DECL E6POS XP287={X 5671.46198,Y -717.1018,Z 4003.704,A -116.65787,B -23.21109,C 16.21129,S 2,T 35,E1 -3867.99764,E2 0,E3 0,E4 0,E5 0,E6 0}
; DECL LDAT LCPDATP147={VEL 1,ACC 100,APO_DIST 100,APO_FAC 50.0,ORI_TYP #VAR,CIRC_TYP #BASE,JERK_FAC 50.0}
DECL FDAT FP288={TOOL_NO 0,BASE_NO 0,IPO_FRAME #BASE,POINT2[] " ",TQ_STATE FALSE}
DECL E6POS XP288={X 12666.37592,Y -538.48386,Z 3708.53974,A -127.07895,B -20.60151,C -3.44033,S 2,T 35,E1 -10812.08896,E2 0,E3 0,E4 0,E5 0,E6 0}
; DECL LDAT LCPDATP113={VEL 1,ACC 100,APO_DIST 100,APO_FAC 50.0,ORI_TYP #VAR,CIRC_TYP #BASE,JERK_FAC 50.0}
DECL FDAT FP289={TOOL_NO 0,BASE_NO 0,IPO_FRAME #BASE,POINT2[] " ",TQ_STATE FALSE}
DECL E6POS XP289={X 6379.94734,Y -681.40788,Z 3158.20554,A -102.40256,B 11.37187,C 4.81103,S 2,T 35,E1 -4209.91162,E2 0,E3 0,E4 0,E5 0,E6 0}
; DECL LDAT LCPDATP114={VEL 1,ACC 100,APO_DIST 100,APO_FAC 50.0,ORI_TYP #VAR,CIRC_TYP #BASE,JERK_FAC 50.0}
DECL FDAT FP290={TOOL_NO 0,BASE_NO 0,IPO_FRAME #BASE,POINT2[] " ",TQ_STATE FALSE}
DECL E6POS XP290={X 6328.481,Y -681.40737,Z 3158.20597,A -102.7078,B 7.77597,C 4.76025,S 2,T 35,E1 -4158.44503,E2 0,E3 0,E4 0,E5 0,E6 0}
; DECL LDAT LCPDATP115={VEL 1,ACC 100,APO_DIST 100,APO_FAC 50.0,ORI_TYP #VAR,CIRC_TYP #BASE,JERK_FAC 50.0}
DECL FDAT FP291={TOOL_NO 0,BASE_NO 0,IPO_FRAME #BASE,POINT2[] " ",TQ_STATE FALSE}
DECL E6POS XP291={X 12929.38089,Y -681.40737,Z 3158.20639,A -83.4604,B -12.81532,C -0.94267,S 2,T 35,E1 -10812.08896,E2 0,E3 0,E4 0,E5 0,E6 0}
; DECL LDAT LCPDATP116={VEL 1,ACC 100,APO_DIST 100,APO_FAC 50.0,ORI_TYP #VAR,CIRC_TYP #BASE,JERK_FAC 50.0}
DECL FDAT FP292={TOOL_NO 0,BASE_NO 0,IPO_FRAME #BASE,POINT2[] " ",TQ_STATE FALSE}
DECL E6POS XP292={X 12886.08572,Y -646.4113,Z 3336.02814,A -83.4604,B -12.81532,C -0.94267,S 2,T 35,E1 -10812.08896,E2 0,E3 0,E4 0,E5 0,E6 0}
; DECL LDAT LCPDATP117={VEL 1,ACC 100,APO_DIST 100,APO_FAC 50.0,ORI_TYP #VAR,CIRC_TYP #BASE,JERK_FAC 50.0}
DECL FDAT FP293={TOOL_NO 0,BASE_NO 0,IPO_FRAME #BASE,POINT2[] " ",TQ_STATE FALSE}
DECL E6POS XP293={X 6226.20694,Y -691.76303,Z 3410.82553,A -102.7078,B 7.77597,C 4.76022,S 2,T 35,E1 -4167.06683,E2 0,E3 0,E4 0,E5 0,E6 0}
; DECL LDAT LCPDATP118={VEL 1,ACC 100,APO_DIST 100,APO_FAC 50.0,ORI_TYP #VAR,CIRC_TYP #BASE,JERK_FAC 50.0}
DECL FDAT FP294={TOOL_NO 0,BASE_NO 0,IPO_FRAME #BASE,POINT2[] " ",TQ_STATE FALSE}
DECL E6POS XP294={X 6109.20944,Y -705.3695,Z 3654.40552,A -102.70779,B 7.77597,C 4.76025,S 2,T 35,E1 -4140.9372,E2 0,E3 0,E4 0,E5 0,E6 0}
; DECL LDAT LCPDATP121={VEL 1,ACC 100,APO_DIST 100,APO_FAC 50.0,ORI_TYP #VAR,CIRC_TYP #BASE,JERK_FAC 50.0}
DECL FDAT FP295={TOOL_NO 0,BASE_NO 0,IPO_FRAME #BASE,POINT2[] " ",TQ_STATE FALSE}
DECL E6POS XP295={X 12777.06723,Y -602.17839,Z 3573.69413,A -83.4604,B -12.81532,C -0.94267,S 2,T 35,E1 -10812.08896,E2 0,E3 0,E4 0,E5 0,E6 0}
; DECL LDAT LCPDATP122={VEL 1,ACC 100,APO_DIST 100,APO_FAC 50.0,ORI_TYP #VAR,CIRC_TYP #BASE,JERK_FAC 50.0}
DECL FDAT FP296={TOOL_NO 0,BASE_NO 0,IPO_FRAME #BASE,POINT2[] " ",TQ_STATE FALSE}
DECL E6POS XP296={X 12675.92788,Y -569.18264,Z 3775.2407,A -83.4604,B -12.81532,C -0.94267,S 2,T 35,E1 -10812.08896,E2 0,E3 0,E4 0,E5 0,E6 0}
; DECL LDAT LCPDATP119={VEL 1,ACC 100,APO_DIST 100,APO_FAC 50.0,ORI_TYP #VAR,CIRC_TYP #BASE,JERK_FAC 50.0}
DECL FDAT FP297={TOOL_NO 0,BASE_NO 0,IPO_FRAME #BASE,POINT2[] " ",TQ_STATE FALSE}
DECL E6POS XP297={X 6034.81499,Y -708.12179,Z 3847.76366,A -102.7078,B 7.77596,C 4.76026,S 2,T 35,E1 -4174.36752,E2 0,E3 0,E4 0,E5 0,E6 0}
; DECL LDAT LCPDATP120={VEL 1,ACC 100,APO_DIST 100,APO_FAC 50.0,ORI_TYP #VAR,CIRC_TYP #BASE,JERK_FAC 50.0}
DECL FDAT FP298={TOOL_NO 0,BASE_NO 0,IPO_FRAME #BASE,POINT2[] " ",TQ_STATE FALSE}
DECL E6POS XP298={X 5808.56571,Y -717.10091,Z 4003.7046,A -102.70779,B 7.77596,C 4.76025,S 2,T 35,E1 -4005.10214,E2 0,E3 0,E4 0,E5 0,E6 0}
; DECL LDAT LCPDATP123={VEL 1,ACC 100,APO_DIST 100,APO_FAC 50.0,ORI_TYP #VAR,CIRC_TYP #BASE,JERK_FAC 50.0}
DECL FDAT FP299={TOOL_NO 0,BASE_NO 0,IPO_FRAME #BASE,POINT2[] " ",TQ_STATE FALSE}
DECL E6POS XP299={X 12607.03936,Y -538.48386,Z 3940.5062,A -83.4604,B -12.81532,C -0.94267,S 2,T 35,E1 -10812.08896,E2 0,E3 0,E4 0,E5 0,E6 0}
; DECL LDAT LCPDATP124={VEL 1,ACC 100,APO_DIST 100,APO_FAC 50.0,ORI_TYP #VAR,CIRC_TYP #BASE,JERK_FAC 50.0}
DECL FDAT FP300={TOOL_NO 0,BASE_NO 0,IPO_FRAME #BASE,POINT2[] " ",TQ_STATE FALSE}
DECL E6POS XP300={X 12329.73693,Y -538.48386,Z 3940.5062,A -83.38777,B -15.32829,C -1.2413,S 2,T 35,E1 -10812.08896,E2 0,E3 0,E4 0,E5 0,E6 0}
; DECL LDAT LCPDATP130={VEL 1,ACC 100,APO_DIST 100,APO_FAC 50.0,ORI_TYP #VAR,CIRC_TYP #BASE,JERK_FAC 50.0}
DECL FDAT FP301={TOOL_NO 0,BASE_NO 0,IPO_FRAME #BASE,POINT2[] " ",TQ_STATE FALSE}
DECL E6POS XP301={X 6035.27715,Y -717.10158,Z 4003.70466,A -106.51042,B 6.34838,C 5.00917,S 2,T 35,E1 -4231.81368,E2 0,E3 0,E4 0,E5 0,E6 0}
; DECL LDAT LCPDATP131={VEL 1,ACC 100,APO_DIST 100,APO_FAC 50.0,ORI_TYP #VAR,CIRC_TYP #BASE,JERK_FAC 50.0}
DECL FDAT FP302={TOOL_NO 0,BASE_NO 0,IPO_FRAME #BASE,POINT2[] " ",TQ_STATE FALSE}
DECL E6POS XP302={X 6001.84737,Y -717.10113,Z 4003.70421,A -106.4599,B 4.5615,C 5.54032,S 2,T 35,E1 -4198.38336,E2 0,E3 0,E4 0,E5 0,E6 0}
; DECL LDAT LCPDATP125={VEL 1,ACC 100,APO_DIST 100,APO_FAC 50.0,ORI_TYP #VAR,CIRC_TYP #BASE,JERK_FAC 50.0}
DECL FDAT FP303={TOOL_NO 0,BASE_NO 0,IPO_FRAME #BASE,POINT2[] " ",TQ_STATE FALSE}
DECL E6POS XP303={X 12327.62864,Y -538.48366,Z 3940.50597,A -87.76623,B -17.49847,C -1.50503,S 2,T 35,E1 -10473.34117,E2 0,E3 0,E4 0,E5 0,E6 0}
; DECL LDAT LCPDATP126={VEL 1,ACC 100,APO_DIST 100,APO_FAC 50.0,ORI_TYP #VAR,CIRC_TYP #BASE,JERK_FAC 50.0}
DECL FDAT FP304={TOOL_NO 0,BASE_NO 0,IPO_FRAME #BASE,POINT2[] " ",TQ_STATE FALSE}
DECL E6POS XP304={X 12344.44126,Y -538.48354,Z 3940.50612,A -92.12133,B -19.55447,C -1.59012,S 2,T 35,E1 -10490.15446,E2 0,E3 0,E4 0,E5 0,E6 0}
; DECL LDAT LCPDATP132={VEL 1,ACC 100,APO_DIST 100,APO_FAC 50.0,ORI_TYP #VAR,CIRC_TYP #BASE,JERK_FAC 50.0}
DECL FDAT FP305={TOOL_NO 0,BASE_NO 0,IPO_FRAME #BASE,POINT2[] " ",TQ_STATE FALSE}
DECL E6POS XP305={X 5984.60315,Y -717.10142,Z 4003.7045,A -107.27293,B 2.66443,C 6.10126,S 2,T 35,E1 -4181.13976,E2 0,E3 0,E4 0,E5 0,E6 0}
; DECL LDAT LCPDATP133={VEL 1,ACC 100,APO_DIST 100,APO_FAC 50.0,ORI_TYP #VAR,CIRC_TYP #BASE,JERK_FAC 50.0}
DECL FDAT FP306={TOOL_NO 0,BASE_NO 0,IPO_FRAME #BASE,POINT2[] " ",TQ_STATE FALSE}
DECL E6POS XP306={X 5959.53065,Y -717.10165,Z 4003.70439,A -107.25516,B 0.74219,C 6.69889,S 2,T 35,E1 -4156.06702,E2 0,E3 0,E4 0,E5 0,E6 0}
; DECL LDAT LCPDATP127={VEL 1,ACC 100,APO_DIST 100,APO_FAC 50.0,ORI_TYP #VAR,CIRC_TYP #BASE,JERK_FAC 50.0}
DECL FDAT FP307={TOOL_NO 0,BASE_NO 0,IPO_FRAME #BASE,POINT2[] " ",TQ_STATE FALSE}
DECL E6POS XP307={X 12327.65948,Y -538.48376,Z 3940.50627,A -96.02004,B -21.56802,C -1.50992,S 2,T 35,E1 -10473.37259,E2 0,E3 0,E4 0,E5 0,E6 0}
; DECL LDAT LCPDATP128={VEL 1,ACC 100,APO_DIST 100,APO_FAC 50.0,ORI_TYP #VAR,CIRC_TYP #BASE,JERK_FAC 50.0}
DECL FDAT FP308={TOOL_NO 0,BASE_NO 0,IPO_FRAME #BASE,POINT2[] " ",TQ_STATE FALSE}
DECL E6POS XP308={X 12434.40962,Y -538.48361,Z 3791.38491,A -100.48203,B -23.59142,C -1.27711,S 2,T 35,E1 -10580.12251,E2 0,E3 0,E4 0,E5 0,E6 0}
; DECL LDAT LCPDATP134={VEL 1,ACC 100,APO_DIST 100,APO_FAC 50.0,ORI_TYP #VAR,CIRC_TYP #BASE,JERK_FAC 50.0}
DECL FDAT FP309={TOOL_NO 0,BASE_NO 0,IPO_FRAME #BASE,POINT2[] " ",TQ_STATE FALSE}
DECL E6POS XP309={X 6027.18413,Y -717.10157,Z 4003.70451,A -108.83879,B -1.2655,C 7.3225,S 2,T 35,E1 -4223.72032,E2 0,E3 0,E4 0,E5 0,E6 0}
; DECL LDAT LCPDATP135={VEL 1,ACC 100,APO_DIST 100,APO_FAC 50.0,ORI_TYP #VAR,CIRC_TYP #BASE,JERK_FAC 50.0}
DECL FDAT FP310={TOOL_NO 0,BASE_NO 0,IPO_FRAME #BASE,POINT2[] " ",TQ_STATE FALSE}
DECL E6POS XP310={X 5994.01853,Y -717.10159,Z 4003.70409,A -109.42003,B -3.44272,C 8.06654,S 2,T 35,E1 -4190.55423,E2 0,E3 0,E4 0,E5 0,E6 0}
; DECL LDAT LCPDATP129={VEL 1,ACC 100,APO_DIST 100,APO_FAC 50.0,ORI_TYP #VAR,CIRC_TYP #BASE,JERK_FAC 50.0}
DECL FDAT FP311={TOOL_NO 0,BASE_NO 0,IPO_FRAME #BASE,POINT2[] " ",TQ_STATE FALSE}
DECL E6POS XP311={X 12525.53957,Y -538.48385,Z 3733.39322,A -103.74147,B -24.12805,C -1.24549,S 2,T 35,E1 -10671.25219,E2 0,E3 0,E4 0,E5 0,E6 0}
; DECL LDAT LCPDATP138={VEL 1,ACC 100,APO_DIST 100,APO_FAC 50.0,ORI_TYP #VAR,CIRC_TYP #BASE,JERK_FAC 50.0}
DECL FDAT FP312={TOOL_NO 0,BASE_NO 0,IPO_FRAME #BASE,POINT2[] " ",TQ_STATE FALSE}
DECL E6POS XP312={X 12409.55634,Y -538.48385,Z 3733.39322,A -103.74147,B -24.12805,C -1.24549,S 2,T 35,E1 -10555.26896,E2 0,E3 0,E4 0,E5 0,E6 0}
; DECL LDAT LCPDATP136={VEL 1,ACC 100,APO_DIST 100,APO_FAC 50.0,ORI_TYP #VAR,CIRC_TYP #BASE,JERK_FAC 50.0}
DECL FDAT FP313={TOOL_NO 0,BASE_NO 0,IPO_FRAME #BASE,POINT2[] " ",TQ_STATE FALSE}
DECL E6POS XP313={X 5960.30101,Y -717.10136,Z 4003.70387,A -109.95564,B -5.51238,C 8.79955,S 2,T 35,E1 -4156.83652,E2 0,E3 0,E4 0,E5 0,E6 0}
; DECL LDAT LCPDATP137={VEL 1,ACC 100,APO_DIST 100,APO_FAC 50.0,ORI_TYP #VAR,CIRC_TYP #BASE,JERK_FAC 50.0}
DECL FDAT FP314={TOOL_NO 0,BASE_NO 0,IPO_FRAME #BASE,POINT2[] " ",TQ_STATE FALSE}
DECL E6POS XP314={X 5959.29294,Y -717.10098,Z 4003.70454,A -110.58224,B -7.77816,C 9.62993,S 2,T 35,E1 -4155.82897,E2 0,E3 0,E4 0,E5 0,E6 0}
; DECL LDAT LCPDATP139={VEL 1,ACC 100,APO_DIST 100,APO_FAC 50.0,ORI_TYP #VAR,CIRC_TYP #BASE,JERK_FAC 50.0}
DECL FDAT FP315={TOOL_NO 0,BASE_NO 0,IPO_FRAME #BASE,POINT2[] " ",TQ_STATE FALSE}
DECL E6POS XP315={X 12666.37592,Y -538.48386,Z 3733.39329,A -110.95703,B -23.34196,C -1.63568,S 2,T 35,E1 -10812.08896,E2 0,E3 0,E4 0,E5 0,E6 0}
; DECL LDAT LCPDATP140={VEL 1,ACC 100,APO_DIST 100,APO_FAC 50.0,ORI_TYP #VAR,CIRC_TYP #BASE,JERK_FAC 50.0}
DECL FDAT FP316={TOOL_NO 0,BASE_NO 0,IPO_FRAME #BASE,POINT2[] " ",TQ_STATE FALSE}
DECL E6POS XP316={X 12666.37592,Y -538.48386,Z 3700.25522,A -113.36831,B -23.34196,C -1.63568,S 2,T 35,E1 -10812.08896,E2 0,E3 0,E4 0,E5 0,E6 0}
; DECL LDAT LCPDATP149={VEL 1,ACC 100,APO_DIST 100,APO_FAC 50.0,ORI_TYP #VAR,CIRC_TYP #BASE,JERK_FAC 50.0}
DECL FDAT FP317={TOOL_NO 0,BASE_NO 0,IPO_FRAME #BASE,POINT2[] " ",TQ_STATE FALSE}
DECL E6POS XP317={X 5916.8006,Y -717.10155,Z 4003.70412,A -110.72224,B -10.13455,C 10.52896,S 2,T 35,E1 -4113.33656,E2 0,E3 0,E4 0,E5 0,E6 0}
; DECL LDAT LCPDATP150={VEL 1,ACC 100,APO_DIST 100,APO_FAC 50.0,ORI_TYP #VAR,CIRC_TYP #BASE,JERK_FAC 50.0}
DECL FDAT FP318={TOOL_NO 0,BASE_NO 0,IPO_FRAME #BASE,POINT2[] " ",TQ_STATE FALSE}
DECL E6POS XP318={X 5875.31565,Y -717.1012,Z 4003.70448,A -110.8879,B -12.32973,C 11.37928,S 2,T 35,E1 -4071.85169,E2 0,E3 0,E4 0,E5 0,E6 0}
; DECL LDAT LCPDATP141={VEL 1,ACC 100,APO_DIST 100,APO_FAC 50.0,ORI_TYP #VAR,CIRC_TYP #BASE,JERK_FAC 50.0}
DECL FDAT FP319={TOOL_NO 0,BASE_NO 0,IPO_FRAME #BASE,POINT2[] " ",TQ_STATE FALSE}
DECL E6POS XP319={X 12666.37592,Y -538.48386,Z 3675.40167,A -115.34787,B -23.34196,C -1.63568,S 2,T 35,E1 -10812.08896,E2 0,E3 0,E4 0,E5 0,E6 0}
; DECL LDAT LCPDATP142={VEL 1,ACC 100,APO_DIST 100,APO_FAC 50.0,ORI_TYP #VAR,CIRC_TYP #BASE,JERK_FAC 50.0}
DECL FDAT FP320={TOOL_NO 0,BASE_NO 0,IPO_FRAME #BASE,POINT2[] " ",TQ_STATE FALSE}
DECL E6POS XP320={X 12666.37592,Y -538.48386,Z 3725.10877,A -117.62399,B -22.31862,C -2.21953,S 2,T 35,E1 -10812.08896,E2 0,E3 0,E4 0,E5 0,E6 0}
; DECL LDAT LCPDATP151={VEL 1,ACC 100,APO_DIST 100,APO_FAC 50.0,ORI_TYP #VAR,CIRC_TYP #BASE,JERK_FAC 50.0}
DECL FDAT FP321={TOOL_NO 0,BASE_NO 0,IPO_FRAME #BASE,POINT2[] " ",TQ_STATE FALSE}
DECL E6POS XP321={X 5898.57722,Y -717.10122,Z 4003.70435,A -112.09203,B -14.38754,C 12.19033,S 2,T 35,E1 -4095.11298,E2 0,E3 0,E4 0,E5 0,E6 0}
; DECL LDAT LCPDATP152={VEL 1,ACC 100,APO_DIST 100,APO_FAC 50.0,ORI_TYP #VAR,CIRC_TYP #BASE,JERK_FAC 50.0}
DECL FDAT FP322={TOOL_NO 0,BASE_NO 0,IPO_FRAME #BASE,POINT2[] " ",TQ_STATE FALSE}
DECL E6POS XP322={X 5854.40488,Y -717.10171,Z 4003.70448,A -112.35649,B -16.71303,C 13.17652,S 2,T 35,E1 -4050.94133,E2 0,E3 0,E4 0,E5 0,E6 0}
; DECL LDAT LCPDATP143={VEL 1,ACC 100,APO_DIST 100,APO_FAC 50.0,ORI_TYP #VAR,CIRC_TYP #BASE,JERK_FAC 50.0}
DECL FDAT FP323={TOOL_NO 0,BASE_NO 0,IPO_FRAME #BASE,POINT2[] " ",TQ_STATE FALSE}
DECL E6POS XP323={X 12666.37592,Y -538.48386,Z 3708.53974,A -119.39266,B -22.0406,C -2.38888,S 2,T 35,E1 -10812.08896,E2 0,E3 0,E4 0,E5 0,E6 0}
; DECL LDAT LCPDATP144={VEL 1,ACC 100,APO_DIST 100,APO_FAC 50.0,ORI_TYP #VAR,CIRC_TYP #BASE,JERK_FAC 50.0}
DECL FDAT FP324={TOOL_NO 0,BASE_NO 0,IPO_FRAME #BASE,POINT2[] " ",TQ_STATE FALSE}
DECL E6POS XP324={X 12666.37592,Y -538.48386,Z 3716.82426,A -121.52366,B -21.70131,C -2.61349,S 2,T 35,E1 -10812.08896,E2 0,E3 0,E4 0,E5 0,E6 0}
; DECL LDAT LCPDATP153={VEL 1,ACC 100,APO_DIST 100,APO_FAC 50.0,ORI_TYP #VAR,CIRC_TYP #BASE,JERK_FAC 50.0}
DECL FDAT FP325={TOOL_NO 0,BASE_NO 0,IPO_FRAME #BASE,POINT2[] " ",TQ_STATE FALSE}
DECL E6POS XP325={X 5865.70091,Y -717.10124,Z 4003.70383,A -113.62634,B -18.80667,C 14.08679,S 2,T 35,E1 -4062.23613,E2 0,E3 0,E4 0,E5 0,E6 0}
; DECL LDAT LCPDATP154={VEL 1,ACC 100,APO_DIST 100,APO_FAC 50.0,ORI_TYP #VAR,CIRC_TYP #BASE,JERK_FAC 50.0}
DECL FDAT FP326={TOOL_NO 0,BASE_NO 0,IPO_FRAME #BASE,POINT2[] " ",TQ_STATE FALSE}
DECL E6POS XP326={X 5786.97193,Y -717.10138,Z 4003.70442,A -113.90846,B -20.59534,C 14.92344,S 2,T 35,E1 -3983.50839,E2 0,E3 0,E4 0,E5 0,E6 0}
; DECL LDAT LCPDATP145={VEL 1,ACC 100,APO_DIST 100,APO_FAC 50.0,ORI_TYP #VAR,CIRC_TYP #BASE,JERK_FAC 50.0}
DECL FDAT FP327={TOOL_NO 0,BASE_NO 0,IPO_FRAME #BASE,POINT2[] " ",TQ_STATE FALSE}
DECL E6POS XP327={X 12666.37592,Y -538.48386,Z 3691.97071,A -122.58569,B -21.70131,C -2.61349,S 2,T 35,E1 -10812.08896,E2 0,E3 0,E4 0,E5 0,E6 0}
; DECL LDAT LCPDATP146={VEL 1,ACC 100,APO_DIST 100,APO_FAC 50.0,ORI_TYP #VAR,CIRC_TYP #BASE,JERK_FAC 50.0}
DECL FDAT FP328={TOOL_NO 0,BASE_NO 0,IPO_FRAME #BASE,POINT2[] " ",TQ_STATE FALSE}
DECL E6POS XP328={X 12666.37592,Y -538.48386,Z 3741.67781,A -124.88801,B -20.60151,C -3.44033,S 2,T 35,E1 -10812.08896,E2 0,E3 0,E4 0,E5 0,E6 0}
; DECL LDAT LCPDATP155={VEL 1,ACC 100,APO_DIST 100,APO_FAC 50.0,ORI_TYP #VAR,CIRC_TYP #BASE,JERK_FAC 50.0}
DECL FDAT FP329={TOOL_NO 0,BASE_NO 0,IPO_FRAME #BASE,POINT2[] " ",TQ_STATE FALSE}
DECL E6POS XP329={X 5766.06143,Y -717.10078,Z 4003.7047,A -114.88478,B -21.82725,C 15.51221,S 2,T 35,E1 -3962.59803,E2 0,E3 0,E4 0,E5 0,E6 0}
; DECL LDAT LCPDATP156={VEL 1,ACC 100,APO_DIST 100,APO_FAC 50.0,ORI_TYP #VAR,CIRC_TYP #BASE,JERK_FAC 50.0}
DECL FDAT FP330={TOOL_NO 0,BASE_NO 0,IPO_FRAME #BASE,POINT2[] " ",TQ_STATE FALSE}
DECL E6POS XP330={X 5671.46198,Y -717.1018,Z 4003.704,A -116.65787,B -23.21109,C 16.21129,S 2,T 35,E1 -3867.99764,E2 0,E3 0,E4 0,E5 0,E6 0}
; DECL LDAT LCPDATP147={VEL 1,ACC 100,APO_DIST 100,APO_FAC 50.0,ORI_TYP #VAR,CIRC_TYP #BASE,JERK_FAC 50.0}
DECL FDAT FP331={TOOL_NO 0,BASE_NO 0,IPO_FRAME #BASE,POINT2[] " ",TQ_STATE FALSE}
DECL E6POS XP331={X 12666.37592,Y -538.48386,Z 3708.53974,A -127.07895,B -20.60151,C -3.44033,S 2,T 35,E1 -10812.08896,E2 0,E3 0,E4 0,E5 0,E6 0}
; DECL LDAT LCPDATP113={VEL 1,ACC 100,APO_DIST 100,APO_FAC 50.0,ORI_TYP #VAR,CIRC_TYP #BASE,JERK_FAC 50.0}
DECL FDAT FP332={TOOL_NO 0,BASE_NO 0,IPO_FRAME #BASE,POINT2[] " ",TQ_STATE FALSE}
DECL E6POS XP332={X 6379.94734,Y -681.40788,Z 3158.20554,A -102.40256,B 11.37187,C 4.81103,S 2,T 35,E1 -4209.91162,E2 0,E3 0,E4 0,E5 0,E6 0}
; DECL LDAT LCPDATP114={VEL 1,ACC 100,APO_DIST 100,APO_FAC 50.0,ORI_TYP #VAR,CIRC_TYP #BASE,JERK_FAC 50.0}
DECL FDAT FP333={TOOL_NO 0,BASE_NO 0,IPO_FRAME #BASE,POINT2[] " ",TQ_STATE FALSE}
DECL E6POS XP333={X 6328.481,Y -681.40737,Z 3158.20597,A -102.7078,B 7.77597,C 4.76025,S 2,T 35,E1 -4158.44503,E2 0,E3 0,E4 0,E5 0,E6 0}
; DECL LDAT LCPDATP115={VEL 1,ACC 100,APO_DIST 100,APO_FAC 50.0,ORI_TYP #VAR,CIRC_TYP #BASE,JERK_FAC 50.0}
DECL FDAT FP334={TOOL_NO 0,BASE_NO 0,IPO_FRAME #BASE,POINT2[] " ",TQ_STATE FALSE}
DECL E6POS XP334={X 12929.38089,Y -681.40737,Z 3158.20639,A -83.4604,B -12.81532,C -0.94267,S 2,T 35,E1 -10812.08896,E2 0,E3 0,E4 0,E5 0,E6 0}
; DECL LDAT LCPDATP116={VEL 1,ACC 100,APO_DIST 100,APO_FAC 50.0,ORI_TYP #VAR,CIRC_TYP #BASE,JERK_FAC 50.0}
DECL FDAT FP335={TOOL_NO 0,BASE_NO 0,IPO_FRAME #BASE,POINT2[] " ",TQ_STATE FALSE}
DECL E6POS XP335={X 12886.08572,Y -646.4113,Z 3336.02814,A -83.4604,B -12.81532,C -0.94267,S 2,T 35,E1 -10812.08896,E2 0,E3 0,E4 0,E5 0,E6 0}
; DECL LDAT LCPDATP117={VEL 1,ACC 100,APO_DIST 100,APO_FAC 50.0,ORI_TYP #VAR,CIRC_TYP #BASE,JERK_FAC 50.0}
DECL FDAT FP336={TOOL_NO 0,BASE_NO 0,IPO_FRAME #BASE,POINT2[] " ",TQ_STATE FALSE}
DECL E6POS XP336={X 6226.20694,Y -691.76303,Z 3410.82553,A -102.7078,B 7.77597,C 4.76022,S 2,T 35,E1 -4167.06683,E2 0,E3 0,E4 0,E5 0,E6 0}
; DECL LDAT LCPDATP118={VEL 1,ACC 100,APO_DIST 100,APO_FAC 50.0,ORI_TYP #VAR,CIRC_TYP #BASE,JERK_FAC 50.0}
DECL FDAT FP337={TOOL_NO 0,BASE_NO 0,IPO_FRAME #BASE,POINT2[] " ",TQ_STATE FALSE}
DECL E6POS XP337={X 6109.20944,Y -705.3695,Z 3654.40552,A -102.70779,B 7.77597,C 4.76025,S 2,T 35,E1 -4140.9372,E2 0,E3 0,E4 0,E5 0,E6 0}
; DECL LDAT LCPDATP121={VEL 1,ACC 100,APO_DIST 100,APO_FAC 50.0,ORI_TYP #VAR,CIRC_TYP #BASE,JERK_FAC 50.0}
DECL FDAT FP338={TOOL_NO 0,BASE_NO 0,IPO_FRAME #BASE,POINT2[] " ",TQ_STATE FALSE}
DECL E6POS XP338={X 12777.06723,Y -602.17839,Z 3573.69413,A -83.4604,B -12.81532,C -0.94267,S 2,T 35,E1 -10812.08896,E2 0,E3 0,E4 0,E5 0,E6 0}
; DECL LDAT LCPDATP122={VEL 1,ACC 100,APO_DIST 100,APO_FAC 50.0,ORI_TYP #VAR,CIRC_TYP #BASE,JERK_FAC 50.0}
DECL FDAT FP339={TOOL_NO 0,BASE_NO 0,IPO_FRAME #BASE,POINT2[] " ",TQ_STATE FALSE}
DECL E6POS XP339={X 12675.92788,Y -569.18264,Z 3775.2407,A -83.4604,B -12.81532,C -0.94267,S 2,T 35,E1 -10812.08896,E2 0,E3 0,E4 0,E5 0,E6 0}
; DECL LDAT LCPDATP119={VEL 1,ACC 100,APO_DIST 100,APO_FAC 50.0,ORI_TYP #VAR,CIRC_TYP #BASE,JERK_FAC 50.0}
DECL FDAT FP340={TOOL_NO 0,BASE_NO 0,IPO_FRAME #BASE,POINT2[] " ",TQ_STATE FALSE}
DECL E6POS XP340={X 6034.81499,Y -708.12179,Z 3847.76366,A -102.7078,B 7.77596,C 4.76026,S 2,T 35,E1 -4174.36752,E2 0,E3 0,E4 0,E5 0,E6 0}
; DECL LDAT LCPDATP120={VEL 1,ACC 100,APO_DIST 100,APO_FAC 50.0,ORI_TYP #VAR,CIRC_TYP #BASE,JERK_FAC 50.0}
DECL FDAT FP341={TOOL_NO 0,BASE_NO 0,IPO_FRAME #BASE,POINT2[] " ",TQ_STATE FALSE}
DECL E6POS XP341={X 5808.56571,Y -717.10091,Z 4003.7046,A -102.70779,B 7.77596,C 4.76025,S 2,T 35,E1 -4005.10214,E2 0,E3 0,E4 0,E5 0,E6 0}
; DECL LDAT LCPDATP123={VEL 1,ACC 100,APO_DIST 100,APO_FAC 50.0,ORI_TYP #VAR,CIRC_TYP #BASE,JERK_FAC 50.0}
DECL FDAT FP342={TOOL_NO 0,BASE_NO 0,IPO_FRAME #BASE,POINT2[] " ",TQ_STATE FALSE}
DECL E6POS XP342={X 12607.03936,Y -538.48386,Z 3940.5062,A -83.4604,B -12.81532,C -0.94267,S 2,T 35,E1 -10812.08896,E2 0,E3 0,E4 0,E5 0,E6 0}
; DECL LDAT LCPDATP124={VEL 1,ACC 100,APO_DIST 100,APO_FAC 50.0,ORI_TYP #VAR,CIRC_TYP #BASE,JERK_FAC 50.0}
DECL FDAT FP343={TOOL_NO 0,BASE_NO 0,IPO_FRAME #BASE,POINT2[] " ",TQ_STATE FALSE}
DECL E6POS XP343={X 12329.73693,Y -538.48386,Z 3940.5062,A -83.38777,B -15.32829,C -1.2413,S 2,T 35,E1 -10812.08896,E2 0,E3 0,E4 0,E5 0,E6 0}
; DECL LDAT LCPDATP130={VEL 1,ACC 100,APO_DIST 100,APO_FAC 50.0,ORI_TYP #VAR,CIRC_TYP #BASE,JERK_FAC 50.0}
DECL FDAT FP344={TOOL_NO 0,BASE_NO 0,IPO_FRAME #BASE,POINT2[] " ",TQ_STATE FALSE}
DECL E6POS XP344={X 6035.27715,Y -717.10158,Z 4003.70466,A -106.51042,B 6.34838,C 5.00917,S 2,T 35,E1 -4231.81368,E2 0,E3 0,E4 0,E5 0,E6 0}
; DECL LDAT LCPDATP131={VEL 1,ACC 100,APO_DIST 100,APO_FAC 50.0,ORI_TYP #VAR,CIRC_TYP #BASE,JERK_FAC 50.0}
DECL FDAT FP345={TOOL_NO 0,BASE_NO 0,IPO_FRAME #BASE,POINT2[] " ",TQ_STATE FALSE}
DECL E6POS XP345={X 6001.84737,Y -717.10113,Z 4003.70421,A -106.4599,B 4.5615,C 5.54032,S 2,T 35,E1 -4198.38336,E2 0,E3 0,E4 0,E5 0,E6 0}
; DECL LDAT LCPDATP125={VEL 1,ACC 100,APO_DIST 100,APO_FAC 50.0,ORI_TYP #VAR,CIRC_TYP #BASE,JERK_FAC 50.0}
DECL FDAT FP346={TOOL_NO 0,BASE_NO 0,IPO_FRAME #BASE,POINT2[] " ",TQ_STATE FALSE}
DECL E6POS XP346={X 12327.62864,Y -538.48366,Z 3940.50597,A -87.76623,B -17.49847,C -1.50503,S 2,T 35,E1 -10473.34117,E2 0,E3 0,E4 0,E5 0,E6 0}
; DECL LDAT LCPDATP126={VEL 1,ACC 100,APO_DIST 100,APO_FAC 50.0,ORI_TYP #VAR,CIRC_TYP #BASE,JERK_FAC 50.0}
DECL FDAT FP347={TOOL_NO 0,BASE_NO 0,IPO_FRAME #BASE,POINT2[] " ",TQ_STATE FALSE}
DECL E6POS XP347={X 12344.44126,Y -538.48354,Z 3940.50612,A -92.12133,B -19.55447,C -1.59012,S 2,T 35,E1 -10490.15446,E2 0,E3 0,E4 0,E5 0,E6 0}
; DECL LDAT LCPDATP132={VEL 1,ACC 100,APO_DIST 100,APO_FAC 50.0,ORI_TYP #VAR,CIRC_TYP #BASE,JERK_FAC 50.0}
DECL FDAT FP348={TOOL_NO 0,BASE_NO 0,IPO_FRAME #BASE,POINT2[] " ",TQ_STATE FALSE}
DECL E6POS XP348={X 5984.60315,Y -717.10142,Z 4003.7045,A -107.27293,B 2.66443,C 6.10126,S 2,T 35,E1 -4181.13976,E2 0,E3 0,E4 0,E5 0,E6 0}
; DECL LDAT LCPDATP133={VEL 1,ACC 100,APO_DIST 100,APO_FAC 50.0,ORI_TYP #VAR,CIRC_TYP #BASE,JERK_FAC 50.0}
DECL FDAT FP349={TOOL_NO 0,BASE_NO 0,IPO_FRAME #BASE,POINT2[] " ",TQ_STATE FALSE}
DECL E6POS XP349={X 5959.53065,Y -717.10165,Z 4003.70439,A -107.25516,B 0.74219,C 6.69889,S 2,T 35,E1 -4156.06702,E2 0,E3 0,E4 0,E5 0,E6 0}
; DECL LDAT LCPDATP127={VEL 1,ACC 100,APO_DIST 100,APO_FAC 50.0,ORI_TYP #VAR,CIRC_TYP #BASE,JERK_FAC 50.0}
DECL FDAT FP350={TOOL_NO 0,BASE_NO 0,IPO_FRAME #BASE,POINT2[] " ",TQ_STATE FALSE}
DECL E6POS XP350={X 12327.65948,Y -538.48376,Z 3940.50627,A -96.02004,B -21.56802,C -1.50992,S 2,T 35,E1 -10473.37259,E2 0,E3 0,E4 0,E5 0,E6 0}
; DECL LDAT LCPDATP128={VEL 1,ACC 100,APO_DIST 100,APO_FAC 50.0,ORI_TYP #VAR,CIRC_TYP #BASE,JERK_FAC 50.0}
DECL FDAT FP351={TOOL_NO 0,BASE_NO 0,IPO_FRAME #BASE,POINT2[] " ",TQ_STATE FALSE}
DECL E6POS XP351={X 12434.40962,Y -538.48361,Z 3791.38491,A -100.48203,B -23.59142,C -1.27711,S 2,T 35,E1 -10580.12251,E2 0,E3 0,E4 0,E5 0,E6 0}
; DECL LDAT LCPDATP134={VEL 1,ACC 100,APO_DIST 100,APO_FAC 50.0,ORI_TYP #VAR,CIRC_TYP #BASE,JERK_FAC 50.0}
DECL FDAT FP352={TOOL_NO 0,BASE_NO 0,IPO_FRAME #BASE,POINT2[] " ",TQ_STATE FALSE}
DECL E6POS XP352={X 6027.18413,Y -717.10157,Z 4003.70451,A -108.83879,B -1.2655,C 7.3225,S 2,T 35,E1 -4223.72032,E2 0,E3 0,E4 0,E5 0,E6 0}
; DECL LDAT LCPDATP135={VEL 1,ACC 100,APO_DIST 100,APO_FAC 50.0,ORI_TYP #VAR,CIRC_TYP #BASE,JERK_FAC 50.0}
DECL FDAT FP353={TOOL_NO 0,BASE_NO 0,IPO_FRAME #BASE,POINT2[] " ",TQ_STATE FALSE}
DECL E6POS XP353={X 5994.01853,Y -717.10159,Z 4003.70409,A -109.42003,B -3.44272,C 8.06654,S 2,T 35,E1 -4190.55423,E2 0,E3 0,E4 0,E5 0,E6 0}
; DECL LDAT LCPDATP129={VEL 1,ACC 100,APO_DIST 100,APO_FAC 50.0,ORI_TYP #VAR,CIRC_TYP #BASE,JERK_FAC 50.0}
DECL FDAT FP354={TOOL_NO 0,BASE_NO 0,IPO_FRAME #BASE,POINT2[] " ",TQ_STATE FALSE}
DECL E6POS XP354={X 12525.53957,Y -538.48385,Z 3733.39322,A -103.74147,B -24.12805,C -1.24549,S 2,T 35,E1 -10671.25219,E2 0,E3 0,E4 0,E5 0,E6 0}
; DECL LDAT LCPDATP138={VEL 1,ACC 100,APO_DIST 100,APO_FAC 50.0,ORI_TYP #VAR,CIRC_TYP #BASE,JERK_FAC 50.0}
DECL FDAT FP355={TOOL_NO 0,BASE_NO 0,IPO_FRAME #BASE,POINT2[] " ",TQ_STATE FALSE}
DECL E6POS XP355={X 12409.55634,Y -538.48385,Z 3733.39322,A -103.74147,B -24.12805,C -1.24549,S 2,T 35,E1 -10555.26896,E2 0,E3 0,E4 0,E5 0,E6 0}
; DECL LDAT LCPDATP136={VEL 1,ACC 100,APO_DIST 100,APO_FAC 50.0,ORI_TYP #VAR,CIRC_TYP #BASE,JERK_FAC 50.0}
DECL FDAT FP356={TOOL_NO 0,BASE_NO 0,IPO_FRAME #BASE,POINT2[] " ",TQ_STATE FALSE}
DECL E6POS XP356={X 5960.30101,Y -717.10136,Z 4003.70387,A -109.95564,B -5.51238,C 8.79955,S 2,T 35,E1 -4156.83652,E2 0,E3 0,E4 0,E5 0,E6 0}
; DECL LDAT LCPDATP137={VEL 1,ACC 100,APO_DIST 100,APO_FAC 50.0,ORI_TYP #VAR,CIRC_TYP #BASE,JERK_FAC 50.0}
DECL FDAT FP357={TOOL_NO 0,BASE_NO 0,IPO_FRAME #BASE,POINT2[] " ",TQ_STATE FALSE}
DECL E6POS XP357={X 5959.29294,Y -717.10098,Z 4003.70454,A -110.58224,B -7.77816,C 9.62993,S 2,T 35,E1 -4155.82897,E2 0,E3 0,E4 0,E5 0,E6 0}
; DECL LDAT LCPDATP139={VEL 1,ACC 100,APO_DIST 100,APO_FAC 50.0,ORI_TYP #VAR,CIRC_TYP #BASE,JERK_FAC 50.0}
DECL FDAT FP358={TOOL_NO 0,BASE_NO 0,IPO_FRAME #BASE,POINT2[] " ",TQ_STATE FALSE}
DECL E6POS XP358={X 12666.37592,Y -538.48386,Z 3733.39329,A -110.95703,B -23.34196,C -1.63568,S 2,T 35,E1 -10812.08896,E2 0,E3 0,E4 0,E5 0,E6 0}
; DECL LDAT LCPDATP140={VEL 1,ACC 100,APO_DIST 100,APO_FAC 50.0,ORI_TYP #VAR,CIRC_TYP #BASE,JERK_FAC 50.0}
DECL FDAT FP359={TOOL_NO 0,BASE_NO 0,IPO_FRAME #BASE,POINT2[] " ",TQ_STATE FALSE}
DECL E6POS XP359={X 12666.37592,Y -538.48386,Z 3700.25522,A -113.36831,B -23.34196,C -1.63568,S 2,T 35,E1 -10812.08896,E2 0,E3 0,E4 0,E5 0,E6 0}
; DECL LDAT LCPDATP149={VEL 1,ACC 100,APO_DIST 100,APO_FAC 50.0,ORI_TYP #VAR,CIRC_TYP #BASE,JERK_FAC 50.0}
DECL FDAT FP360={TOOL_NO 0,BASE_NO 0,IPO_FRAME #BASE,POINT2[] " ",TQ_STATE FALSE}
DECL E6POS XP360={X 5916.8006,Y -717.10155,Z 4003.70412,A -110.72224,B -10.13455,C 10.52896,S 2,T 35,E1 -4113.33656,E2 0,E3 0,E4 0,E5 0,E6 0}
; DECL LDAT LCPDATP150={VEL 1,ACC 100,APO_DIST 100,APO_FAC 50.0,ORI_TYP #VAR,CIRC_TYP #BASE,JERK_FAC 50.0}
DECL FDAT FP361={TOOL_NO 0,BASE_NO 0,IPO_FRAME #BASE,POINT2[] " ",TQ_STATE FALSE}
DECL E6POS XP361={X 5875.31565,Y -717.1012,Z 4003.70448,A -110.8879,B -12.32973,C 11.37928,S 2,T 35,E1 -4071.85169,E2 0,E3 0,E4 0,E5 0,E6 0}
; DECL LDAT LCPDATP141={VEL 1,ACC 100,APO_DIST 100,APO_FAC 50.0,ORI_TYP #VAR,CIRC_TYP #BASE,JERK_FAC 50.0}
DECL FDAT FP362={TOOL_NO 0,BASE_NO 0,IPO_FRAME #BASE,POINT2[] " ",TQ_STATE FALSE}
DECL E6POS XP362={X 12666.37592,Y -538.48386,Z 3675.40167,A -115.34787,B -23.34196,C -1.63568,S 2,T 35,E1 -10812.08896,E2 0,E3 0,E4 0,E5 0,E6 0}
; DECL LDAT LCPDATP142={VEL 1,ACC 100,APO_DIST 100,APO_FAC 50.0,ORI_TYP #VAR,CIRC_TYP #BASE,JERK_FAC 50.0}
DECL FDAT FP363={TOOL_NO 0,BASE_NO 0,IPO_FRAME #BASE,POINT2[] " ",TQ_STATE FALSE}
DECL E6POS XP363={X 12666.37592,Y -538.48386,Z 3725.10877,A -117.62399,B -22.31862,C -2.21953,S 2,T 35,E1 -10812.08896,E2 0,E3 0,E4 0,E5 0,E6 0}
; DECL LDAT LCPDATP151={VEL 1,ACC 100,APO_DIST 100,APO_FAC 50.0,ORI_TYP #VAR,CIRC_TYP #BASE,JERK_FAC 50.0}
DECL FDAT FP364={TOOL_NO 0,BASE_NO 0,IPO_FRAME #BASE,POINT2[] " ",TQ_STATE FALSE}
DECL E6POS XP364={X 5898.57722,Y -717.10122,Z 4003.70435,A -112.09203,B -14.38754,C 12.19033,S 2,T 35,E1 -4095.11298,E2 0,E3 0,E4 0,E5 0,E6 0}
; DECL LDAT LCPDATP152={VEL 1,ACC 100,APO_DIST 100,APO_FAC 50.0,ORI_TYP #VAR,CIRC_TYP #BASE,JERK_FAC 50.0}
DECL FDAT FP365={TOOL_NO 0,BASE_NO 0,IPO_FRAME #BASE,POINT2[] " ",TQ_STATE FALSE}
DECL E6POS XP365={X 5854.40488,Y -717.10171,Z 4003.70448,A -112.35649,B -16.71303,C 13.17652,S 2,T 35,E1 -4050.94133,E2 0,E3 0,E4 0,E5 0,E6 0}
; DECL LDAT LCPDATP143={VEL 1,ACC 100,APO_DIST 100,APO_FAC 50.0,ORI_TYP #VAR,CIRC_TYP #BASE,JERK_FAC 50.0}
DECL FDAT FP366={TOOL_NO 0,BASE_NO 0,IPO_FRAME #BASE,POINT2[] " ",TQ_STATE FALSE}
DECL E6POS XP366={X 12666.37592,Y -538.48386,Z 3708.53974,A -119.39266,B -22.0406,C -2.38888,S 2,T 35,E1 -10812.08896,E2 0,E3 0,E4 0,E5 0,E6 0}
; DECL LDAT LCPDATP144={VEL 1,ACC 100,APO_DIST 100,APO_FAC 50.0,ORI_TYP #VAR,CIRC_TYP #BASE,JERK_FAC 50.0}
DECL FDAT FP367={TOOL_NO 0,BASE_NO 0,IPO_FRAME #BASE,POINT2[] " ",TQ_STATE FALSE}
DECL E6POS XP367={X 12666.37592,Y -538.48386,Z 3716.82426,A -121.52366,B -21.70131,C -2.61349,S 2,T 35,E1 -10812.08896,E2 0,E3 0,E4 0,E5 0,E6 0}
; DECL LDAT LCPDATP153={VEL 1,ACC 100,APO_DIST 100,APO_FAC 50.0,ORI_TYP #VAR,CIRC_TYP #BASE,JERK_FAC 50.0}
DECL FDAT FP368={TOOL_NO 0,BASE_NO 0,IPO_FRAME #BASE,POINT2[] " ",TQ_STATE FALSE}
DECL E6POS XP368={X 5865.70091,Y -717.10124,Z 4003.70383,A -113.62634,B -18.80667,C 14.08679,S 2,T 35,E1 -4062.23613,E2 0,E3 0,E4 0,E5 0,E6 0}
; DECL LDAT LCPDATP154={VEL 1,ACC 100,APO_DIST 100,APO_FAC 50.0,ORI_TYP #VAR,CIRC_TYP #BASE,JERK_FAC 50.0}
DECL FDAT FP369={TOOL_NO 0,BASE_NO 0,IPO_FRAME #BASE,POINT2[] " ",TQ_STATE FALSE}
DECL E6POS XP369={X 5786.97193,Y -717.10138,Z 4003.70442,A -113.90846,B -20.59534,C 14.92344,S 2,T 35,E1 -3983.50839,E2 0,E3 0,E4 0,E5 0,E6 0}
; DECL LDAT LCPDATP145={VEL 1,ACC 100,APO_DIST 100,APO_FAC 50.0,ORI_TYP #VAR,CIRC_TYP #BASE,JERK_FAC 50.0}
DECL FDAT FP370={TOOL_NO 0,BASE_NO 0,IPO_FRAME #BASE,POINT2[] " ",TQ_STATE FALSE}
DECL E6POS XP370={X 12666.37592,Y -538.48386,Z 3691.97071,A -122.58569,B -21.70131,C -2.61349,S 2,T 35,E1 -10812.08896,E2 0,E3 0,E4 0,E5 0,E6 0}
; DECL LDAT LCPDATP146={VEL 1,ACC 100,APO_DIST 100,APO_FAC 50.0,ORI_TYP #VAR,CIRC_TYP #BASE,JERK_FAC 50.0}
DECL FDAT FP371={TOOL_NO 0,BASE_NO 0,IPO_FRAME #BASE,POINT2[] " ",TQ_STATE FALSE}
DECL E6POS XP371={X 12666.37592,Y -538.48386,Z 3741.67781,A -124.88801,B -20.60151,C -3.44033,S 2,T 35,E1 -10812.08896,E2 0,E3 0,E4 0,E5 0,E6 0}
; DECL LDAT LCPDATP155={VEL 1,ACC 100,APO_DIST 100,APO_FAC 50.0,ORI_TYP #VAR,CIRC_TYP #BASE,JERK_FAC 50.0}
DECL FDAT FP372={TOOL_NO 0,BASE_NO 0,IPO_FRAME #BASE,POINT2[] " ",TQ_STATE FALSE}
DECL E6POS XP372={X 5766.06143,Y -717.10078,Z 4003.7047,A -114.88478,B -21.82725,C 15.51221,S 2,T 35,E1 -3962.59803,E2 0,E3 0,E4 0,E5 0,E6 0}
; DECL LDAT LCPDATP156={VEL 1,ACC 100,APO_DIST 100,APO_FAC 50.0,ORI_TYP #VAR,CIRC_TYP #BASE,JERK_FAC 50.0}
DECL FDAT FP373={TOOL_NO 0,BASE_NO 0,IPO_FRAME #BASE,POINT2[] " ",TQ_STATE FALSE}
DECL E6POS XP373={X 5671.46198,Y -717.1018,Z 4003.704,A -116.65787,B -23.21109,C 16.21129,S 2,T 35,E1 -3867.99764,E2 0,E3 0,E4 0,E5 0,E6 0}
; DECL LDAT LCPDATP147={VEL 1,ACC 100,APO_DIST 100,APO_FAC 50.0,ORI_TYP #VAR,CIRC_TYP #BASE,JERK_FAC 50.0}
DECL FDAT FP374={TOOL_NO 0,BASE_NO 0,IPO_FRAME #BASE,POINT2[] " ",TQ_STATE FALSE}
DECL E6POS XP374={X 12666.37592,Y -538.48386,Z 3708.53974,A -127.07895,B -20.60151,C -3.44033,S 2,T 35,E1 -10812.08896,E2 0,E3 0,E4 0,E5 0,E6 0}
; DECL LDAT LCPDATP113={VEL 1,ACC 100,APO_DIST 100,APO_FAC 50.0,ORI_TYP #VAR,CIRC_TYP #BASE,JERK_FAC 50.0}
DECL FDAT FP375={TOOL_NO 0,BASE_NO 0,IPO_FRAME #BASE,POINT2[] " ",TQ_STATE FALSE}
DECL E6POS XP375={X 6379.94734,Y -681.40788,Z 3158.20554,A -102.40256,B 11.37187,C 4.81103,S 2,T 35,E1 -4209.91162,E2 0,E3 0,E4 0,E5 0,E6 0}
; DECL LDAT LCPDATP114={VEL 1,ACC 100,APO_DIST 100,APO_FAC 50.0,ORI_TYP #VAR,CIRC_TYP #BASE,JERK_FAC 50.0}
DECL FDAT FP376={TOOL_NO 0,BASE_NO 0,IPO_FRAME #BASE,POINT2[] " ",TQ_STATE FALSE}
DECL E6POS XP376={X 6328.481,Y -681.40737,Z 3158.20597,A -102.7078,B 7.77597,C 4.76025,S 2,T 35,E1 -4158.44503,E2 0,E3 0,E4 0,E5 0,E6 0}
; DECL LDAT LCPDATP115={VEL 1,ACC 100,APO_DIST 100,APO_FAC 50.0,ORI_TYP #VAR,CIRC_TYP #BASE,JERK_FAC 50.0}
DECL FDAT FP377={TOOL_NO 0,BASE_NO 0,IPO_FRAME #BASE,POINT2[] " ",TQ_STATE FALSE}
DECL E6POS XP377={X 12929.38089,Y -681.40737,Z 3158.20639,A -83.4604,B -12.81532,C -0.94267,S 2,T 35,E1 -10812.08896,E2 0,E3 0,E4 0,E5 0,E6 0}
; DECL LDAT LCPDATP116={VEL 1,ACC 100,APO_DIST 100,APO_FAC 50.0,ORI_TYP #VAR,CIRC_TYP #BASE,JERK_FAC 50.0}
DECL FDAT FP378={TOOL_NO 0,BASE_NO 0,IPO_FRAME #BASE,POINT2[] " ",TQ_STATE FALSE}
DECL E6POS XP378={X 12886.08572,Y -646.4113,Z 3336.02814,A -83.4604,B -12.81532,C -0.94267,S 2,T 35,E1 -10812.08896,E2 0,E3 0,E4 0,E5 0,E6 0}
; DECL LDAT LCPDATP117={VEL 1,ACC 100,APO_DIST 100,APO_FAC 50.0,ORI_TYP #VAR,CIRC_TYP #BASE,JERK_FAC 50.0}
DECL FDAT FP379={TOOL_NO 0,BASE_NO 0,IPO_FRAME #BASE,POINT2[] " ",TQ_STATE FALSE}
DECL E6POS XP379={X 6226.20694,Y -691.76303,Z 3410.82553,A -102.7078,B 7.77597,C 4.76022,S 2,T 35,E1 -4167.06683,E2 0,E3 0,E4 0,E5 0,E6 0}
; DECL LDAT LCPDATP118={VEL 1,ACC 100,APO_DIST 100,APO_FAC 50.0,ORI_TYP #VAR,CIRC_TYP #BASE,JERK_FAC 50.0}
DECL FDAT FP380={TOOL_NO 0,BASE_NO 0,IPO_FRAME #BASE,POINT2[] " ",TQ_STATE FALSE}
DECL E6POS XP380={X 6109.20944,Y -705.3695,Z 3654.40552,A -102.70779,B 7.77597,C 4.76025,S 2,T 35,E1 -4140.9372,E2 0,E3 0,E4 0,E5 0,E6 0}
; DECL LDAT LCPDATP121={VEL 1,ACC 100,APO_DIST 100,APO_FAC 50.0,ORI_TYP #VAR,CIRC_TYP #BASE,JERK_FAC 50.0}
DECL FDAT FP381={TOOL_NO 0,BASE_NO 0,IPO_FRAME #BASE,POINT2[] " ",TQ_STATE FALSE}
DECL E6POS XP381={X 12777.06723,Y -602.17839,Z 3573.69413,A -83.4604,B -12.81532,C -0.94267,S 2,T 35,E1 -10812.08896,E2 0,E3 0,E4 0,E5 0,E6 0}
; DECL LDAT LCPDATP122={VEL 1,ACC 100,APO_DIST 100,APO_FAC 50.0,ORI_TYP #VAR,CIRC_TYP #BASE,JERK_FAC 50.0}
DECL FDAT FP382={TOOL_NO 0,BASE_NO 0,IPO_FRAME #BASE,POINT2[] " ",TQ_STATE FALSE}
DECL E6POS XP382={X 12675.92788,Y -569.18264,Z 3775.2407,A -83.4604,B -12.81532,C -0.94267,S 2,T 35,E1 -10812.08896,E2 0,E3 0,E4 0,E5 0,E6 0}
; DECL LDAT LCPDATP119={VEL 1,ACC 100,APO_DIST 100,APO_FAC 50.0,ORI_TYP #VAR,CIRC_TYP #BASE,JERK_FAC 50.0}
DECL FDAT FP383={TOOL_NO 0,BASE_NO 0,IPO_FRAME #BASE,POINT2[] " ",TQ_STATE FALSE}
DECL E6POS XP383={X 6034.81499,Y -708.12179,Z 3847.76366,A -102.7078,B 7.77596,C 4.76026,S 2,T 35,E1 -4174.36752,E2 0,E3 0,E4 0,E5 0,E6 0}
; DECL LDAT LCPDATP120={VEL 1,ACC 100,APO_DIST 100,APO_FAC 50.0,ORI_TYP #VAR,CIRC_TYP #BASE,JERK_FAC 50.0}
DECL FDAT FP384={TOOL_NO 0,BASE_NO 0,IPO_FRAME #BASE,POINT2[] " ",TQ_STATE FALSE}
DECL E6POS XP384={X 5808.56571,Y -717.10091,Z 4003.7046,A -102.70779,B 7.77596,C 4.76025,S 2,T 35,E1 -4005.10214,E2 0,E3 0,E4 0,E5 0,E6 0}
; DECL LDAT LCPDATP123={VEL 1,ACC 100,APO_DIST 100,APO_FAC 50.0,ORI_TYP #VAR,CIRC_TYP #BASE,JERK_FAC 50.0}
DECL FDAT FP385={TOOL_NO 0,BASE_NO 0,IPO_FRAME #BASE,POINT2[] " ",TQ_STATE FALSE}
DECL E6POS XP385={X 12607.03936,Y -538.48386,Z 3940.5062,A -83.4604,B -12.81532,C -0.94267,S 2,T 35,E1 -10812.08896,E2 0,E3 0,E4 0,E5 0,E6 0}
; DECL LDAT LCPDATP124={VEL 1,ACC 100,APO_DIST 100,APO_FAC 50.0,ORI_TYP #VAR,CIRC_TYP #BASE,JERK_FAC 50.0}
DECL FDAT FP386={TOOL_NO 0,BASE_NO 0,IPO_FRAME #BASE,POINT2[] " ",TQ_STATE FALSE}
DECL E6POS XP386={X 12329.73693,Y -538.48386,Z 3940.5062,A -83.38777,B -15.32829,C -1.2413,S 2,T 35,E1 -10812.08896,E2 0,E3 0,E4 0,E5 0,E6 0}
; DECL LDAT LCPDATP130={VEL 1,ACC 100,APO_DIST 100,APO_FAC 50.0,ORI_TYP #VAR,CIRC_TYP #BASE,JERK_FAC 50.0}
DECL FDAT FP387={TOOL_NO 0,BASE_NO 0,IPO_FRAME #BASE,POINT2[] " ",TQ_STATE FALSE}
DECL E6POS XP387={X 6035.27715,Y -717.10158,Z 4003.70466,A -106.51042,B 6.34838,C 5.00917,S 2,T 35,E1 -4231.81368,E2 0,E3 0,E4 0,E5 0,E6 0}
; DECL LDAT LCPDATP131={VEL 1,ACC 100,APO_DIST 100,APO_FAC 50.0,ORI_TYP #VAR,CIRC_TYP #BASE,JERK_FAC 50.0}
DECL FDAT FP388={TOOL_NO 0,BASE_NO 0,IPO_FRAME #BASE,POINT2[] " ",TQ_STATE FALSE}
DECL E6POS XP388={X 6001.84737,Y -717.10113,Z 4003.70421,A -106.4599,B 4.5615,C 5.54032,S 2,T 35,E1 -4198.38336,E2 0,E3 0,E4 0,E5 0,E6 0}
; DECL LDAT LCPDATP125={VEL 1,ACC 100,APO_DIST 100,APO_FAC 50.0,ORI_TYP #VAR,CIRC_TYP #BASE,JERK_FAC 50.0}
DECL FDAT FP389={TOOL_NO 0,BASE_NO 0,IPO_FRAME #BASE,POINT2[] " ",TQ_STATE FALSE}
DECL E6POS XP389={X 12327.62864,Y -538.48366,Z 3940.50597,A -87.76623,B -17.49847,C -1.50503,S 2,T 35,E1 -10473.34117,E2 0,E3 0,E4 0,E5 0,E6 0}
; DECL LDAT LCPDATP126={VEL 1,ACC 100,APO_DIST 100,APO_FAC 50.0,ORI_TYP #VAR,CIRC_TYP #BASE,JERK_FAC 50.0}
DECL FDAT FP390={TOOL_NO 0,BASE_NO 0,IPO_FRAME #BASE,POINT2[] " ",TQ_STATE FALSE}
DECL E6POS XP390={X 12344.44126,Y -538.48354,Z 3940.50612,A -92.12133,B -19.55447,C -1.59012,S 2,T 35,E1 -10490.15446,E2 0,E3 0,E4 0,E5 0,E6 0}
; DECL LDAT LCPDATP132={VEL 1,ACC 100,APO_DIST 100,APO_FAC 50.0,ORI_TYP #VAR,CIRC_TYP #BASE,JERK_FAC 50.0}
DECL FDAT FP391={TOOL_NO 0,BASE_NO 0,IPO_FRAME #BASE,POINT2[] " ",TQ_STATE FALSE}
DECL E6POS XP391={X 5984.60315,Y -717.10142,Z 4003.7045,A -107.27293,B 2.66443,C 6.10126,S 2,T 35,E1 -4181.13976,E2 0,E3 0,E4 0,E5 0,E6 0}
; DECL LDAT LCPDATP133={VEL 1,ACC 100,APO_DIST 100,APO_FAC 50.0,ORI_TYP #VAR,CIRC_TYP #BASE,JERK_FAC 50.0}
DECL FDAT FP392={TOOL_NO 0,BASE_NO 0,IPO_FRAME #BASE,POINT2[] " ",TQ_STATE FALSE}
DECL E6POS XP392={X 5959.53065,Y -717.10165,Z 4003.70439,A -107.25516,B 0.74219,C 6.69889,S 2,T 35,E1 -4156.06702,E2 0,E3 0,E4 0,E5 0,E6 0}
; DECL LDAT LCPDATP127={VEL 1,ACC 100,APO_DIST 100,APO_FAC 50.0,ORI_TYP #VAR,CIRC_TYP #BASE,JERK_FAC 50.0}
DECL FDAT FP393={TOOL_NO 0,BASE_NO 0,IPO_FRAME #BASE,POINT2[] " ",TQ_STATE FALSE}
DECL E6POS XP393={X 12327.65948,Y -538.48376,Z 3940.50627,A -96.02004,B -21.56802,C -1.50992,S 2,T 35,E1 -10473.37259,E2 0,E3 0,E4 0,E5 0,E6 0}
; DECL LDAT LCPDATP128={VEL 1,ACC 100,APO_DIST 100,APO_FAC 50.0,ORI_TYP #VAR,CIRC_TYP #BASE,JERK_FAC 50.0}
DECL FDAT FP394={TOOL_NO 0,BASE_NO 0,IPO_FRAME #BASE,POINT2[] " ",TQ_STATE FALSE}
DECL E6POS XP394={X 12434.40962,Y -538.48361,Z 3791.38491,A -100.48203,B -23.59142,C -1.27711,S 2,T 35,E1 -10580.12251,E2 0,E3 0,E4 0,E5 0,E6 0}
; DECL LDAT LCPDATP134={VEL 1,ACC 100,APO_DIST 100,APO_FAC 50.0,ORI_TYP #VAR,CIRC_TYP #BASE,JERK_FAC 50.0}
DECL FDAT FP395={TOOL_NO 0,BASE_NO 0,IPO_FRAME #BASE,POINT2[] " ",TQ_STATE FALSE}
DECL E6POS XP395={X 6027.18413,Y -717.10157,Z 4003.70451,A -108.83879,B -1.2655,C 7.3225,S 2,T 35,E1 -4223.72032,E2 0,E3 0,E4 0,E5 0,E6 0}
; DECL LDAT LCPDATP135={VEL 1,ACC 100,APO_DIST 100,APO_FAC 50.0,ORI_TYP #VAR,CIRC_TYP #BASE,JERK_FAC 50.0}
DECL FDAT FP396={TOOL_NO 0,BASE_NO 0,IPO_FRAME #BASE,POINT2[] " ",TQ_STATE FALSE}
DECL E6POS XP396={X 5994.01853,Y -717.10159,Z 4003.70409,A -109.42003,B -3.44272,C 8.06654,S 2,T 35,E1 -4190.55423,E2 0,E3 0,E4 0,E5 0,E6 0}
; DECL LDAT LCPDATP129={VEL 1,ACC 100,APO_DIST 100,APO_FAC 50.0,ORI_TYP #VAR,CIRC_TYP #BASE,JERK_FAC 50.0}
DECL FDAT FP397={TOOL_NO 0,BASE_NO 0,IPO_FRAME #BASE,POINT2[] " ",TQ_STATE FALSE}
DECL E6POS XP397={X 12525.53957,Y -538.48385,Z 3733.39322,A -103.74147,B -24.12805,C -1.24549,S 2,T 35,E1 -10671.25219,E2 0,E3 0,E4 0,E5 0,E6 0}
; DECL LDAT LCPDATP138={VEL 1,ACC 100,APO_DIST 100,APO_FAC 50.0,ORI_TYP #VAR,CIRC_TYP #BASE,JERK_FAC 50.0}
DECL FDAT FP398={TOOL_NO 0,BASE_NO 0,IPO_FRAME #BASE,POINT2[] " ",TQ_STATE FALSE}
DECL E6POS XP398={X 12409.55634,Y -538.48385,Z 3733.39322,A -103.74147,B -24.12805,C -1.24549,S 2,T 35,E1 -10555.26896,E2 0,E3 0,E4 0,E5 0,E6 0}
; DECL LDAT LCPDATP136={VEL 1,ACC 100,APO_DIST 100,APO_FAC 50.0,ORI_TYP #VAR,CIRC_TYP #BASE,JERK_FAC 50.0}
DECL FDAT FP399={TOOL_NO 0,BASE_NO 0,IPO_FRAME #BASE,POINT2[] " ",TQ_STATE FALSE}
DECL E6POS XP399={X 5960.30101,Y -717.10136,Z 4003.70387,A -109.95564,B -5.51238,C 8.79955,S 2,T 35,E1 -4156.83652,E2 0,E3 0,E4 0,E5 0,E6 0}
; DECL LDAT LCPDATP137={VEL 1,ACC 100,APO_DIST 100,APO_FAC 50.0,ORI_TYP #VAR,CIRC_TYP #BASE,JERK_FAC 50.0}
DECL FDAT FP400={TOOL_NO 0,BASE_NO 0,IPO_FRAME #BASE,POINT2[] " ",TQ_STATE FALSE}
DECL E6POS XP400={X 5959.29294,Y -717.10098,Z 4003.70454,A -110.58224,B -7.77816,C 9.62993,S 2,T 35,E1 -4155.82897,E2 0,E3 0,E4 0,E5 0,E6 0}
; DECL LDAT LCPDATP139={VEL 1,ACC 100,APO_DIST 100,APO_FAC 50.0,ORI_TYP #VAR,CIRC_TYP #BASE,JERK_FAC 50.0}
DECL FDAT FP401={TOOL_NO 0,BASE_NO 0,IPO_FRAME #BASE,POINT2[] " ",TQ_STATE FALSE}
DECL E6POS XP401={X 12666.37592,Y -538.48386,Z 3733.39329,A -110.95703,B -23.34196,C -1.63568,S 2,T 35,E1 -10812.08896,E2 0,E3 0,E4 0,E5 0,E6 0}
; DECL LDAT LCPDATP140={VEL 1,ACC 100,APO_DIST 100,APO_FAC 50.0,ORI_TYP #VAR,CIRC_TYP #BASE,JERK_FAC 50.0}
DECL FDAT FP402={TOOL_NO 0,BASE_NO 0,IPO_FRAME #BASE,POINT2[] " ",TQ_STATE FALSE}
DECL E6POS XP402={X 12666.37592,Y -538.48386,Z 3700.25522,A -113.36831,B -23.34196,C -1.63568,S 2,T 35,E1 -10812.08896,E2 0,E3 0,E4 0,E5 0,E6 0}
; DECL LDAT LCPDATP149={VEL 1,ACC 100,APO_DIST 100,APO_FAC 50.0,ORI_TYP #VAR,CIRC_TYP #BASE,JERK_FAC 50.0}
DECL FDAT FP403={TOOL_NO 0,BASE_NO 0,IPO_FRAME #BASE,POINT2[] " ",TQ_STATE FALSE}
DECL E6POS XP403={X 5916.8006,Y -717.10155,Z 4003.70412,A -110.72224,B -10.13455,C 10.52896,S 2,T 35,E1 -4113.33656,E2 0,E3 0,E4 0,E5 0,E6 0}
; DECL LDAT LCPDATP150={VEL 1,ACC 100,APO_DIST 100,APO_FAC 50.0,ORI_TYP #VAR,CIRC_TYP #BASE,JERK_FAC 50.0}
DECL FDAT FP404={TOOL_NO 0,BASE_NO 0,IPO_FRAME #BASE,POINT2[] " ",TQ_STATE FALSE}
DECL E6POS XP404={X 5875.31565,Y -717.1012,Z 4003.70448,A -110.8879,B -12.32973,C 11.37928,S 2,T 35,E1 -4071.85169,E2 0,E3 0,E4 0,E5 0,E6 0}
; DECL LDAT LCPDATP141={VEL 1,ACC 100,APO_DIST 100,APO_FAC 50.0,ORI_TYP #VAR,CIRC_TYP #BASE,JERK_FAC 50.0}
DECL FDAT FP405={TOOL_NO 0,BASE_NO 0,IPO_FRAME #BASE,POINT2[] " ",TQ_STATE FALSE}
DECL E6POS XP405={X 12666.37592,Y -538.48386,Z 3675.40167,A -115.34787,B -23.34196,C -1.63568,S 2,T 35,E1 -10812.08896,E2 0,E3 0,E4 0,E5 0,E6 0}
; DECL LDAT LCPDATP142={VEL 1,ACC 100,APO_DIST 100,APO_FAC 50.0,ORI_TYP #VAR,CIRC_TYP #BASE,JERK_FAC 50.0}
DECL FDAT FP406={TOOL_NO 0,BASE_NO 0,IPO_FRAME #BASE,POINT2[] " ",TQ_STATE FALSE}
DECL E6POS XP406={X 12666.37592,Y -538.48386,Z 3725.10877,A -117.62399,B -22.31862,C -2.21953,S 2,T 35,E1 -10812.08896,E2 0,E3 0,E4 0,E5 0,E6 0}
; DECL LDAT LCPDATP151={VEL 1,ACC 100,APO_DIST 100,APO_FAC 50.0,ORI_TYP #VAR,CIRC_TYP #BASE,JERK_FAC 50.0}
DECL FDAT FP407={TOOL_NO 0,BASE_NO 0,IPO_FRAME #BASE,POINT2[] " ",TQ_STATE FALSE}
DECL E6POS XP407={X 5898.57722,Y -717.10122,Z 4003.70435,A -112.09203,B -14.38754,C 12.19033,S 2,T 35,E1 -4095.11298,E2 0,E3 0,E4 0,E5 0,E6 0}
; DECL LDAT LCPDATP152={VEL 1,ACC 100,APO_DIST 100,APO_FAC 50.0,ORI_TYP #VAR,CIRC_TYP #BASE,JERK_FAC 50.0}
DECL FDAT FP408={TOOL_NO 0,BASE_NO 0,IPO_FRAME #BASE,POINT2[] " ",TQ_STATE FALSE}
DECL E6POS XP408={X 5854.40488,Y -717.10171,Z 4003.70448,A -112.35649,B -16.71303,C 13.17652,S 2,T 35,E1 -4050.94133,E2 0,E3 0,E4 0,E5 0,E6 0}
; DECL LDAT LCPDATP143={VEL 1,ACC 100,APO_DIST 100,APO_FAC 50.0,ORI_TYP #VAR,CIRC_TYP #BASE,JERK_FAC 50.0}
DECL FDAT FP409={TOOL_NO 0,BASE_NO 0,IPO_FRAME #BASE,POINT2[] " ",TQ_STATE FALSE}
DECL E6POS XP409={X 12666.37592,Y -538.48386,Z 3708.53974,A -119.39266,B -22.0406,C -2.38888,S 2,T 35,E1 -10812.08896,E2 0,E3 0,E4 0,E5 0,E6 0}
; DECL LDAT LCPDATP144={VEL 1,ACC 100,APO_DIST 100,APO_FAC 50.0,ORI_TYP #VAR,CIRC_TYP #BASE,JERK_FAC 50.0}
DECL FDAT FP410={TOOL_NO 0,BASE_NO 0,IPO_FRAME #BASE,POINT2[] " ",TQ_STATE FALSE}
DECL E6POS XP410={X 12666.37592,Y -538.48386,Z 3716.82426,A -121.52366,B -21.70131,C -2.61349,S 2,T 35,E1 -10812.08896,E2 0,E3 0,E4 0,E5 0,E6 0}
; DECL LDAT LCPDATP153={VEL 1,ACC 100,APO_DIST 100,APO_FAC 50.0,ORI_TYP #VAR,CIRC_TYP #BASE,JERK_FAC 50.0}
DECL FDAT FP411={TOOL_NO 0,BASE_NO 0,IPO_FRAME #BASE,POINT2[] " ",TQ_STATE FALSE}
DECL E6POS XP411={X 5865.70091,Y -717.10124,Z 4003.70383,A -113.62634,B -18.80667,C 14.08679,S 2,T 35,E1 -4062.23613,E2 0,E3 0,E4 0,E5 0,E6 0}
; DECL LDAT LCPDATP154={VEL 1,ACC 100,APO_DIST 100,APO_FAC 50.0,ORI_TYP #VAR,CIRC_TYP #BASE,JERK_FAC 50.0}
DECL FDAT FP412={TOOL_NO 0,BASE_NO 0,IPO_FRAME #BASE,POINT2[] " ",TQ_STATE FALSE}
DECL E6POS XP412={X 5786.97193,Y -717.10138,Z 4003.70442,A -113.90846,B -20.59534,C 14.92344,S 2,T 35,E1 -3983.50839,E2 0,E3 0,E4 0,E5 0,E6 0}
; DECL LDAT LCPDATP145={VEL 1,ACC 100,APO_DIST 100,APO_FAC 50.0,ORI_TYP #VAR,CIRC_TYP #BASE,JERK_FAC 50.0}
DECL FDAT FP413={TOOL_NO 0,BASE_NO 0,IPO_FRAME #BASE,POINT2[] " ",TQ_STATE FALSE}
DECL E6POS XP413={X 12666.37592,Y -538.48386,Z 3691.97071,A -122.58569,B -21.70131,C -2.61349,S 2,T 35,E1 -10812.08896,E2 0,E3 0,E4 0,E5 0,E6 0}
; DECL LDAT LCPDATP146={VEL 1,ACC 100,APO_DIST 100,APO_FAC 50.0,ORI_TYP #VAR,CIRC_TYP #BASE,JERK_FAC 50.0}
DECL FDAT FP414={TOOL_NO 0,BASE_NO 0,IPO_FRAME #BASE,POINT2[] " ",TQ_STATE FALSE}
DECL E6POS XP414={X 12666.37592,Y -538.48386,Z 3741.67781,A -124.88801,B -20.60151,C -3.44033,S 2,T 35,E1 -10812.08896,E2 0,E3 0,E4 0,E5 0,E6 0}
; DECL LDAT LCPDATP155={VEL 1,ACC 100,APO_DIST 100,APO_FAC 50.0,ORI_TYP #VAR,CIRC_TYP #BASE,JERK_FAC 50.0}
DECL FDAT FP415={TOOL_NO 0,BASE_NO 0,IPO_FRAME #BASE,POINT2[] " ",TQ_STATE FALSE}
DECL E6POS XP415={X 5766.06143,Y -717.10078,Z 4003.7047,A -114.88478,B -21.82725,C 15.51221,S 2,T 35,E1 -3962.59803,E2 0,E3 0,E4 0,E5 0,E6 0}
; DECL LDAT LCPDATP156={VEL 1,ACC 100,APO_DIST 100,APO_FAC 50.0,ORI_TYP #VAR,CIRC_TYP #BASE,JERK_FAC 50.0}
DECL FDAT FP416={TOOL_NO 0,BASE_NO 0,IPO_FRAME #BASE,POINT2[] " ",TQ_STATE FALSE}
DECL E6POS XP416={X 5671.46198,Y -717.1018,Z 4003.704,A -116.65787,B -23.21109,C 16.21129,S 2,T 35,E1 -3867.99764,E2 0,E3 0,E4 0,E5 0,E6 0}
; DECL LDAT LCPDATP147={VEL 1,ACC 100,APO_DIST 100,APO_FAC 50.0,ORI_TYP #VAR,CIRC_TYP #BASE,JERK_FAC 50.0}
DECL FDAT FP417={TOOL_NO 0,BASE_NO 0,IPO_FRAME #BASE,POINT2[] " ",TQ_STATE FALSE}
DECL E6POS XP417={X 12666.37592,Y -538.48386,Z 3708.53974,A -127.07895,B -20.60151,C -3.44033,S 2,T 35,E1 -10812.08896,E2 0,E3 0,E4 0,E5 0,E6 0}
; DECL LDAT LCPDATP113={VEL 1,ACC 100,APO_DIST 100,APO_FAC 50.0,ORI_TYP #VAR,CIRC_TYP #BASE,JERK_FAC 50.0}
DECL FDAT FP418={TOOL_NO 0,BASE_NO 0,IPO_FRAME #BASE,POINT2[] " ",TQ_STATE FALSE}
DECL E6POS XP418={X 6379.94734,Y -681.40788,Z 3158.20554,A -102.40256,B 11.37187,C 4.81103,S 2,T 35,E1 -4209.91162,E2 0,E3 0,E4 0,E5 0,E6 0}
; DECL LDAT LCPDATP114={VEL 1,ACC 100,APO_DIST 100,APO_FAC 50.0,ORI_TYP #VAR,CIRC_TYP #BASE,JERK_FAC 50.0}
DECL FDAT FP419={TOOL_NO 0,BASE_NO 0,IPO_FRAME #BASE,POINT2[] " ",TQ_STATE FALSE}
DECL E6POS XP419={X 6328.481,Y -681.40737,Z 3158.20597,A -102.7078,B 7.77597,C 4.76025,S 2,T 35,E1 -4158.44503,E2 0,E3 0,E4 0,E5 0,E6 0}
; DECL LDAT LCPDATP115={VEL 1,ACC 100,APO_DIST 100,APO_FAC 50.0,ORI_TYP #VAR,CIRC_TYP #BASE,JERK_FAC 50.0}
DECL FDAT FP420={TOOL_NO 0,BASE_NO 0,IPO_FRAME #BASE,POINT2[] " ",TQ_STATE FALSE}
DECL E6POS XP420={X 12929.38089,Y -681.40737,Z 3158.20639,A -83.4604,B -12.81532,C -0.94267,S 2,T 35,E1 -10812.08896,E2 0,E3 0,E4 0,E5 0,E6 0}
; DECL LDAT LCPDATP116={VEL 1,ACC 100,APO_DIST 100,APO_FAC 50.0,ORI_TYP #VAR,CIRC_TYP #BASE,JERK_FAC 50.0}
DECL FDAT FP421={TOOL_NO 0,BASE_NO 0,IPO_FRAME #BASE,POINT2[] " ",TQ_STATE FALSE}
DECL E6POS XP421={X 12886.08572,Y -646.4113,Z 3336.02814,A -83.4604,B -12.81532,C -0.94267,S 2,T 35,E1 -10812.08896,E2 0,E3 0,E4 0,E5 0,E6 0}
; DECL LDAT LCPDATP117={VEL 1,ACC 100,APO_DIST 100,APO_FAC 50.0,ORI_TYP #VAR,CIRC_TYP #BASE,JERK_FAC 50.0}
DECL FDAT FP422={TOOL_NO 0,BASE_NO 0,IPO_FRAME #BASE,POINT2[] " ",TQ_STATE FALSE}
DECL E6POS XP422={X 6226.20694,Y -691.76303,Z 3410.82553,A -102.7078,B 7.77597,C 4.76022,S 2,T 35,E1 -4167.06683,E2 0,E3 0,E4 0,E5 0,E6 0}
; DECL LDAT LCPDATP118={VEL 1,ACC 100,APO_DIST 100,APO_FAC 50.0,ORI_TYP #VAR,CIRC_TYP #BASE,JERK_FAC 50.0}
DECL FDAT FP423={TOOL_NO 0,BASE_NO 0,IPO_FRAME #BASE,POINT2[] " ",TQ_STATE FALSE}
DECL E6POS XP423={X 6109.20944,Y -705.3695,Z 3654.40552,A -102.70779,B 7.77597,C 4.76025,S 2,T 35,E1 -4140.9372,E2 0,E3 0,E4 0,E5 0,E6 0}
; DECL LDAT LCPDATP121={VEL 1,ACC 100,APO_DIST 100,APO_FAC 50.0,ORI_TYP #VAR,CIRC_TYP #BASE,JERK_FAC 50.0}
DECL FDAT FP424={TOOL_NO 0,BASE_NO 0,IPO_FRAME #BASE,POINT2[] " ",TQ_STATE FALSE}
DECL E6POS XP424={X 12777.06723,Y -602.17839,Z 3573.69413,A -83.4604,B -12.81532,C -0.94267,S 2,T 35,E1 -10812.08896,E2 0,E3 0,E4 0,E5 0,E6 0}
; DECL LDAT LCPDATP122={VEL 1,ACC 100,APO_DIST 100,APO_FAC 50.0,ORI_TYP #VAR,CIRC_TYP #BASE,JERK_FAC 50.0}
DECL FDAT FP425={TOOL_NO 0,BASE_NO 0,IPO_FRAME #BASE,POINT2[] " ",TQ_STATE FALSE}
DECL E6POS XP425={X 12675.92788,Y -569.18264,Z 3775.2407,A -83.4604,B -12.81532,C -0.94267,S 2,T 35,E1 -10812.08896,E2 0,E3 0,E4 0,E5 0,E6 0}
; DECL LDAT LCPDATP119={VEL 1,ACC 100,APO_DIST 100,APO_FAC 50.0,ORI_TYP #VAR,CIRC_TYP #BASE,JERK_FAC 50.0}
DECL FDAT FP426={TOOL_NO 0,BASE_NO 0,IPO_FRAME #BASE,POINT2[] " ",TQ_STATE FALSE}
DECL E6POS XP426={X 6034.81499,Y -708.12179,Z 3847.76366,A -102.7078,B 7.77596,C 4.76026,S 2,T 35,E1 -4174.36752,E2 0,E3 0,E4 0,E5 0,E6 0}
; DECL LDAT LCPDATP120={VEL 1,ACC 100,APO_DIST 100,APO_FAC 50.0,ORI_TYP #VAR,CIRC_TYP #BASE,JERK_FAC 50.0}
DECL FDAT FP427={TOOL_NO 0,BASE_NO 0,IPO_FRAME #BASE,POINT2[] " ",TQ_STATE FALSE}
DECL E6POS XP427={X 5808.56571,Y -717.10091,Z 4003.7046,A -102.70779,B 7.77596,C 4.76025,S 2,T 35,E1 -4005.10214,E2 0,E3 0,E4 0,E5 0,E6 0}
; DECL LDAT LCPDATP123={VEL 1,ACC 100,APO_DIST 100,APO_FAC 50.0,ORI_TYP #VAR,CIRC_TYP #BASE,JERK_FAC 50.0}
DECL FDAT FP428={TOOL_NO 0,BASE_NO 0,IPO_FRAME #BASE,POINT2[] " ",TQ_STATE FALSE}
DECL E6POS XP428={X 12607.03936,Y -538.48386,Z 3940.5062,A -83.4604,B -12.81532,C -0.94267,S 2,T 35,E1 -10812.08896,E2 0,E3 0,E4 0,E5 0,E6 0}
; DECL LDAT LCPDATP124={VEL 1,ACC 100,APO_DIST 100,APO_FAC 50.0,ORI_TYP #VAR,CIRC_TYP #BASE,JERK_FAC 50.0}
DECL FDAT FP429={TOOL_NO 0,BASE_NO 0,IPO_FRAME #BASE,POINT2[] " ",TQ_STATE FALSE}
DECL E6POS XP429={X 12329.73693,Y -538.48386,Z 3940.5062,A -83.38777,B -15.32829,C -1.2413,S 2,T 35,E1 -10812.08896,E2 0,E3 0,E4 0,E5 0,E6 0}
; DECL LDAT LCPDATP130={VEL 1,ACC 100,APO_DIST 100,APO_FAC 50.0,ORI_TYP #VAR,CIRC_TYP #BASE,JERK_FAC 50.0}
DECL FDAT FP430={TOOL_NO 0,BASE_NO 0,IPO_FRAME #BASE,POINT2[] " ",TQ_STATE FALSE}
DECL E6POS XP430={X 6035.27715,Y -717.10158,Z 4003.70466,A -106.51042,B 6.34838,C 5.00917,S 2,T 35,E1 -4231.81368,E2 0,E3 0,E4 0,E5 0,E6 0}
; DECL LDAT LCPDATP131={VEL 1,ACC 100,APO_DIST 100,APO_FAC 50.0,ORI_TYP #VAR,CIRC_TYP #BASE,JERK_FAC 50.0}
DECL FDAT FP431={TOOL_NO 0,BASE_NO 0,IPO_FRAME #BASE,POINT2[] " ",TQ_STATE FALSE}
DECL E6POS XP431={X 6001.84737,Y -717.10113,Z 4003.70421,A -106.4599,B 4.5615,C 5.54032,S 2,T 35,E1 -4198.38336,E2 0,E3 0,E4 0,E5 0,E6 0}
; DECL LDAT LCPDATP125={VEL 1,ACC 100,APO_DIST 100,APO_FAC 50.0,ORI_TYP #VAR,CIRC_TYP #BASE,JERK_FAC 50.0}
DECL FDAT FP432={TOOL_NO 0,BASE_NO 0,IPO_FRAME #BASE,POINT2[] " ",TQ_STATE FALSE}
DECL E6POS XP432={X 12327.62864,Y -538.48366,Z 3940.50597,A -87.76623,B -17.49847,C -1.50503,S 2,T 35,E1 -10473.34117,E2 0,E3 0,E4 0,E5 0,E6 0}
; DECL LDAT LCPDATP126={VEL 1,ACC 100,APO_DIST 100,APO_FAC 50.0,ORI_TYP #VAR,CIRC_TYP #BASE,JERK_FAC 50.0}
DECL FDAT FP433={TOOL_NO 0,BASE_NO 0,IPO_FRAME #BASE,POINT2[] " ",TQ_STATE FALSE}
DECL E6POS XP433={X 12344.44126,Y -538.48354,Z 3940.50612,A -92.12133,B -19.55447,C -1.59012,S 2,T 35,E1 -10490.15446,E2 0,E3 0,E4 0,E5 0,E6 0}
; DECL LDAT LCPDATP132={VEL 1,ACC 100,APO_DIST 100,APO_FAC 50.0,ORI_TYP #VAR,CIRC_TYP #BASE,JERK_FAC 50.0}
DECL FDAT FP434={TOOL_NO 0,BASE_NO 0,IPO_FRAME #BASE,POINT2[] " ",TQ_STATE FALSE}
DECL E6POS XP434={X 5984.60315,Y -717.10142,Z 4003.7045,A -107.27293,B 2.66443,C 6.10126,S 2,T 35,E1 -4181.13976,E2 0,E3 0,E4 0,E5 0,E6 0}
; DECL LDAT LCPDATP133={VEL 1,ACC 100,APO_DIST 100,APO_FAC 50.0,ORI_TYP #VAR,CIRC_TYP #BASE,JERK_FAC 50.0}
DECL FDAT FP435={TOOL_NO 0,BASE_NO 0,IPO_FRAME #BASE,POINT2[] " ",TQ_STATE FALSE}
DECL E6POS XP435={X 5959.53065,Y -717.10165,Z 4003.70439,A -107.25516,B 0.74219,C 6.69889,S 2,T 35,E1 -4156.06702,E2 0,E3 0,E4 0,E5 0,E6 0}
; DECL LDAT LCPDATP127={VEL 1,ACC 100,APO_DIST 100,APO_FAC 50.0,ORI_TYP #VAR,CIRC_TYP #BASE,JERK_FAC 50.0}
DECL FDAT FP436={TOOL_NO 0,BASE_NO 0,IPO_FRAME #BASE,POINT2[] " ",TQ_STATE FALSE}
DECL E6POS XP436={X 12327.65948,Y -538.48376,Z 3940.50627,A -96.02004,B -21.56802,C -1.50992,S 2,T 35,E1 -10473.37259,E2 0,E3 0,E4 0,E5 0,E6 0}
; DECL LDAT LCPDATP128={VEL 1,ACC 100,APO_DIST 100,APO_FAC 50.0,ORI_TYP #VAR,CIRC_TYP #BASE,JERK_FAC 50.0}
DECL FDAT FP437={TOOL_NO 0,BASE_NO 0,IPO_FRAME #BASE,POINT2[] " ",TQ_STATE FALSE}
DECL E6POS XP437={X 12434.40962,Y -538.48361,Z 3791.38491,A -100.48203,B -23.59142,C -1.27711,S 2,T 35,E1 -10580.12251,E2 0,E3 0,E4 0,E5 0,E6 0}
; DECL LDAT LCPDATP134={VEL 1,ACC 100,APO_DIST 100,APO_FAC 50.0,ORI_TYP #VAR,CIRC_TYP #BASE,JERK_FAC 50.0}
DECL FDAT FP438={TOOL_NO 0,BASE_NO 0,IPO_FRAME #BASE,POINT2[] " ",TQ_STATE FALSE}
DECL E6POS XP438={X 6027.18413,Y -717.10157,Z 4003.70451,A -108.83879,B -1.2655,C 7.3225,S 2,T 35,E1 -4223.72032,E2 0,E3 0,E4 0,E5 0,E6 0}
; DECL LDAT LCPDATP135={VEL 1,ACC 100,APO_DIST 100,APO_FAC 50.0,ORI_TYP #VAR,CIRC_TYP #BASE,JERK_FAC 50.0}
DECL FDAT FP439={TOOL_NO 0,BASE_NO 0,IPO_FRAME #BASE,POINT2[] " ",TQ_STATE FALSE}
DECL E6POS XP439={X 5994.01853,Y -717.10159,Z 4003.70409,A -109.42003,B -3.44272,C 8.06654,S 2,T 35,E1 -4190.55423,E2 0,E3 0,E4 0,E5 0,E6 0}
; DECL LDAT LCPDATP129={VEL 1,ACC 100,APO_DIST 100,APO_FAC 50.0,ORI_TYP #VAR,CIRC_TYP #BASE,JERK_FAC 50.0}
DECL FDAT FP440={TOOL_NO 0,BASE_NO 0,IPO_FRAME #BASE,POINT2[] " ",TQ_STATE FALSE}
DECL E6POS XP440={X 12525.53957,Y -538.48385,Z 3733.39322,A -103.74147,B -24.12805,C -1.24549,S 2,T 35,E1 -10671.25219,E2 0,E3 0,E4 0,E5 0,E6 0}
; DECL LDAT LCPDATP138={VEL 1,ACC 100,APO_DIST 100,APO_FAC 50.0,ORI_TYP #VAR,CIRC_TYP #BASE,JERK_FAC 50.0}
DECL FDAT FP441={TOOL_NO 0,BASE_NO 0,IPO_FRAME #BASE,POINT2[] " ",TQ_STATE FALSE}
DECL E6POS XP441={X 12409.55634,Y -538.48385,Z 3733.39322,A -103.74147,B -24.12805,C -1.24549,S 2,T 35,E1 -10555.26896,E2 0,E3 0,E4 0,E5 0,E6 0}
; DECL LDAT LCPDATP136={VEL 1,ACC 100,APO_DIST 100,APO_FAC 50.0,ORI_TYP #VAR,CIRC_TYP #BASE,JERK_FAC 50.0}
DECL FDAT FP442={TOOL_NO 0,BASE_NO 0,IPO_FRAME #BASE,POINT2[] " ",TQ_STATE FALSE}
DECL E6POS XP442={X 5960.30101,Y -717.10136,Z 4003.70387,A -109.95564,B -5.51238,C 8.79955,S 2,T 35,E1 -4156.83652,E2 0,E3 0,E4 0,E5 0,E6 0}
; DECL LDAT LCPDATP137={VEL 1,ACC 100,APO_DIST 100,APO_FAC 50.0,ORI_TYP #VAR,CIRC_TYP #BASE,JERK_FAC 50.0}
DECL FDAT FP443={TOOL_NO 0,BASE_NO 0,IPO_FRAME #BASE,POINT2[] " ",TQ_STATE FALSE}
DECL E6POS XP443={X 5959.29294,Y -717.10098,Z 4003.70454,A -110.58224,B -7.77816,C 9.62993,S 2,T 35,E1 -4155.82897,E2 0,E3 0,E4 0,E5 0,E6 0}
; DECL LDAT LCPDATP139={VEL 1,ACC 100,APO_DIST 100,APO_FAC 50.0,ORI_TYP #VAR,CIRC_TYP #BASE,JERK_FAC 50.0}
DECL FDAT FP444={TOOL_NO 0,BASE_NO 0,IPO_FRAME #BASE,POINT2[] " ",TQ_STATE FALSE}
DECL E6POS XP444={X 12666.37592,Y -538.48386,Z 3733.39329,A -110.95703,B -23.34196,C -1.63568,S 2,T 35,E1 -10812.08896,E2 0,E3 0,E4 0,E5 0,E6 0}
; DECL LDAT LCPDATP140={VEL 1,ACC 100,APO_DIST 100,APO_FAC 50.0,ORI_TYP #VAR,CIRC_TYP #BASE,JERK_FAC 50.0}
DECL FDAT FP445={TOOL_NO 0,BASE_NO 0,IPO_FRAME #BASE,POINT2[] " ",TQ_STATE FALSE}
DECL E6POS XP445={X 12666.37592,Y -538.48386,Z 3700.25522,A -113.36831,B -23.34196,C -1.63568,S 2,T 35,E1 -10812.08896,E2 0,E3 0,E4 0,E5 0,E6 0}
; DECL LDAT LCPDATP149={VEL 1,ACC 100,APO_DIST 100,APO_FAC 50.0,ORI_TYP #VAR,CIRC_TYP #BASE,JERK_FAC 50.0}
DECL FDAT FP446={TOOL_NO 0,BASE_NO 0,IPO_FRAME #BASE,POINT2[] " ",TQ_STATE FALSE}
DECL E6POS XP446={X 5916.8006,Y -717.10155,Z 4003.70412,A -110.72224,B -10.13455,C 10.52896,S 2,T 35,E1 -4113.33656,E2 0,E3 0,E4 0,E5 0,E6 0}
; DECL LDAT LCPDATP150={VEL 1,ACC 100,APO_DIST 100,APO_FAC 50.0,ORI_TYP #VAR,CIRC_TYP #BASE,JERK_FAC 50.0}
DECL FDAT FP447={TOOL_NO 0,BASE_NO 0,IPO_FRAME #BASE,POINT2[] " ",TQ_STATE FALSE}
DECL E6POS XP447={X 5875.31565,Y -717.1012,Z 4003.70448,A -110.8879,B -12.32973,C 11.37928,S 2,T 35,E1 -4071.85169,E2 0,E3 0,E4 0,E5 0,E6 0}
; DECL LDAT LCPDATP141={VEL 1,ACC 100,APO_DIST 100,APO_FAC 50.0,ORI_TYP #VAR,CIRC_TYP #BASE,JERK_FAC 50.0}
DECL FDAT FP448={TOOL_NO 0,BASE_NO 0,IPO_FRAME #BASE,POINT2[] " ",TQ_STATE FALSE}
DECL E6POS XP448={X 12666.37592,Y -538.48386,Z 3675.40167,A -115.34787,B -23.34196,C -1.63568,S 2,T 35,E1 -10812.08896,E2 0,E3 0,E4 0,E5 0,E6 0}
; DECL LDAT LCPDATP142={VEL 1,ACC 100,APO_DIST 100,APO_FAC 50.0,ORI_TYP #VAR,CIRC_TYP #BASE,JERK_FAC 50.0}
DECL FDAT FP449={TOOL_NO 0,BASE_NO 0,IPO_FRAME #BASE,POINT2[] " ",TQ_STATE FALSE}
DECL E6POS XP449={X 12666.37592,Y -538.48386,Z 3725.10877,A -117.62399,B -22.31862,C -2.21953,S 2,T 35,E1 -10812.08896,E2 0,E3 0,E4 0,E5 0,E6 0}
; DECL LDAT LCPDATP151={VEL 1,ACC 100,APO_DIST 100,APO_FAC 50.0,ORI_TYP #VAR,CIRC_TYP #BASE,JERK_FAC 50.0}
DECL FDAT FP450={TOOL_NO 0,BASE_NO 0,IPO_FRAME #BASE,POINT2[] " ",TQ_STATE FALSE}
DECL E6POS XP450={X 5898.57722,Y -717.10122,Z 4003.70435,A -112.09203,B -14.38754,C 12.19033,S 2,T 35,E1 -4095.11298,E2 0,E3 0,E4 0,E5 0,E6 0}
; DECL LDAT LCPDATP152={VEL 1,ACC 100,APO_DIST 100,APO_FAC 50.0,ORI_TYP #VAR,CIRC_TYP #BASE,JERK_FAC 50.0}
DECL FDAT FP451={TOOL_NO 0,BASE_NO 0,IPO_FRAME #BASE,POINT2[] " ",TQ_STATE FALSE}
DECL E6POS XP451={X 5854.40488,Y -717.10171,Z 4003.70448,A -112.35649,B -16.71303,C 13.17652,S 2,T 35,E1 -4050.94133,E2 0,E3 0,E4 0,E5 0,E6 0}
; DECL LDAT LCPDATP143={VEL 1,ACC 100,APO_DIST 100,APO_FAC 50.0,ORI_TYP #VAR,CIRC_TYP #BASE,JERK_FAC 50.0}
DECL FDAT FP452={TOOL_NO 0,BASE_NO 0,IPO_FRAME #BASE,POINT2[] " ",TQ_STATE FALSE}
DECL E6POS XP452={X 12666.37592,Y -538.48386,Z 3708.53974,A -119.39266,B -22.0406,C -2.38888,S 2,T 35,E1 -10812.08896,E2 0,E3 0,E4 0,E5 0,E6 0}
; DECL LDAT LCPDATP144={VEL 1,ACC 100,APO_DIST 100,APO_FAC 50.0,ORI_TYP #VAR,CIRC_TYP #BASE,JERK_FAC 50.0}
DECL FDAT FP453={TOOL_NO 0,BASE_NO 0,IPO_FRAME #BASE,POINT2[] " ",TQ_STATE FALSE}
DECL E6POS XP453={X 12666.37592,Y -538.48386,Z 3716.82426,A -121.52366,B -21.70131,C -2.61349,S 2,T 35,E1 -10812.08896,E2 0,E3 0,E4 0,E5 0,E6 0}
; DECL LDAT LCPDATP153={VEL 1,ACC 100,APO_DIST 100,APO_FAC 50.0,ORI_TYP #VAR,CIRC_TYP #BASE,JERK_FAC 50.0}
DECL FDAT FP454={TOOL_NO 0,BASE_NO 0,IPO_FRAME #BASE,POINT2[] " ",TQ_STATE FALSE}
DECL E6POS XP454={X 5865.70091,Y -717.10124,Z 4003.70383,A -113.62634,B -18.80667,C 14.08679,S 2,T 35,E1 -4062.23613,E2 0,E3 0,E4 0,E5 0,E6 0}
; DECL LDAT LCPDATP154={VEL 1,ACC 100,APO_DIST 100,APO_FAC 50.0,ORI_TYP #VAR,CIRC_TYP #BASE,JERK_FAC 50.0}
DECL FDAT FP455={TOOL_NO 0,BASE_NO 0,IPO_FRAME #BASE,POINT2[] " ",TQ_STATE FALSE}
DECL E6POS XP455={X 5786.97193,Y -717.10138,Z 4003.70442,A -113.90846,B -20.59534,C 14.92344,S 2,T 35,E1 -3983.50839,E2 0,E3 0,E4 0,E5 0,E6 0}
; DECL LDAT LCPDATP145={VEL 1,ACC 100,APO_DIST 100,APO_FAC 50.0,ORI_TYP #VAR,CIRC_TYP #BASE,JERK_FAC 50.0}
DECL FDAT FP456={TOOL_NO 0,BASE_NO 0,IPO_FRAME #BASE,POINT2[] " ",TQ_STATE FALSE}
DECL E6POS XP456={X 12666.37592,Y -538.48386,Z 3691.97071,A -122.58569,B -21.70131,C -2.61349,S 2,T 35,E1 -10812.08896,E2 0,E3 0,E4 0,E5 0,E6 0}
; DECL LDAT LCPDATP146={VEL 1,ACC 100,APO_DIST 100,APO_FAC 50.0,ORI_TYP #VAR,CIRC_TYP #BASE,JERK_FAC 50.0}
DECL FDAT FP457={TOOL_NO 0,BASE_NO 0,IPO_FRAME #BASE,POINT2[] " ",TQ_STATE FALSE}
DECL E6POS XP457={X 12666.37592,Y -538.48386,Z 3741.67781,A -124.88801,B -20.60151,C -3.44033,S 2,T 35,E1 -10812.08896,E2 0,E3 0,E4 0,E5 0,E6 0}
; DECL LDAT LCPDATP155={VEL 1,ACC 100,APO_DIST 100,APO_FAC 50.0,ORI_TYP #VAR,CIRC_TYP #BASE,JERK_FAC 50.0}
DECL FDAT FP458={TOOL_NO 0,BASE_NO 0,IPO_FRAME #BASE,POINT2[] " ",TQ_STATE FALSE}
DECL E6POS XP458={X 5766.06143,Y -717.10078,Z 4003.7047,A -114.88478,B -21.82725,C 15.51221,S 2,T 35,E1 -3962.59803,E2 0,E3 0,E4 0,E5 0,E6 0}
; DECL LDAT LCPDATP156={VEL 1,ACC 100,APO_DIST 100,APO_FAC 50.0,ORI_TYP #VAR,CIRC_TYP #BASE,JERK_FAC 50.0}
DECL FDAT FP459={TOOL_NO 0,BASE_NO 0,IPO_FRAME #BASE,POINT2[] " ",TQ_STATE FALSE}
DECL E6POS XP459={X 5671.46198,Y -717.1018,Z 4003.704,A -116.65787,B -23.21109,C 16.21129,S 2,T 35,E1 -3867.99764,E2 0,E3 0,E4 0,E5 0,E6 0}
; DECL LDAT LCPDATP147={VEL 1,ACC 100,APO_DIST 100,APO_FAC 50.0,ORI_TYP #VAR,CIRC_TYP #BASE,JERK_FAC 50.0}
DECL FDAT FP460={TOOL_NO 0,BASE_NO 0,IPO_FRAME #BASE,POINT2[] " ",TQ_STATE FALSE}
DECL E6POS XP460={X 12666.37592,Y -538.48386,Z 3708.53974,A -127.07895,B -20.60151,C -3.44033,S 2,T 35,E1 -10812.08896,E2 0,E3 0,E4 0,E5 0,E6 0}
; DECL LDAT LCPDATP113={VEL 1,ACC 100,APO_DIST 100,APO_FAC 50.0,ORI_TYP #VAR,CIRC_TYP #BASE,JERK_FAC 50.0}
DECL FDAT FP461={TOOL_NO 0,BASE_NO 0,IPO_FRAME #BASE,POINT2[] " ",TQ_STATE FALSE}
DECL E6POS XP461={X 6379.94734,Y -681.40788,Z 3158.20554,A -102.40256,B 11.37187,C 4.81103,S 2,T 35,E1 -4209.91162,E2 0,E3 0,E4 0,E5 0,E6 0}
; DECL LDAT LCPDATP114={VEL 1,ACC 100,APO_DIST 100,APO_FAC 50.0,ORI_TYP #VAR,CIRC_TYP #BASE,JERK_FAC 50.0}
DECL FDAT FP462={TOOL_NO 0,BASE_NO 0,IPO_FRAME #BASE,POINT2[] " ",TQ_STATE FALSE}
DECL E6POS XP462={X 6328.481,Y -681.40737,Z 3158.20597,A -102.7078,B 7.77597,C 4.76025,S 2,T 35,E1 -4158.44503,E2 0,E3 0,E4 0,E5 0,E6 0}
; DECL LDAT LCPDATP115={VEL 1,ACC 100,APO_DIST 100,APO_FAC 50.0,ORI_TYP #VAR,CIRC_TYP #BASE,JERK_FAC 50.0}
DECL FDAT FP463={TOOL_NO 0,BASE_NO 0,IPO_FRAME #BASE,POINT2[] " ",TQ_STATE FALSE}
DECL E6POS XP463={X 12929.38089,Y -681.40737,Z 3158.20639,A -83.4604,B -12.81532,C -0.94267,S 2,T 35,E1 -10812.08896,E2 0,E3 0,E4 0,E5 0,E6 0}
; DECL LDAT LCPDATP116={VEL 1,ACC 100,APO_DIST 100,APO_FAC 50.0,ORI_TYP #VAR,CIRC_TYP #BASE,JERK_FAC 50.0}
DECL FDAT FP464={TOOL_NO 0,BASE_NO 0,IPO_FRAME #BASE,POINT2[] " ",TQ_STATE FALSE}
DECL E6POS XP464={X 12886.08572,Y -646.4113,Z 3336.02814,A -83.4604,B -12.81532,C -0.94267,S 2,T 35,E1 -10812.08896,E2 0,E3 0,E4 0,E5 0,E6 0}
; DECL LDAT LCPDATP117={VEL 1,ACC 100,APO_DIST 100,APO_FAC 50.0,ORI_TYP #VAR,CIRC_TYP #BASE,JERK_FAC 50.0}
DECL FDAT FP465={TOOL_NO 0,BASE_NO 0,IPO_FRAME #BASE,POINT2[] " ",TQ_STATE FALSE}
DECL E6POS XP465={X 6226.20694,Y -691.76303,Z 3410.82553,A -102.7078,B 7.77597,C 4.76022,S 2,T 35,E1 -4167.06683,E2 0,E3 0,E4 0,E5 0,E6 0}
; DECL LDAT LCPDATP118={VEL 1,ACC 100,APO_DIST 100,APO_FAC 50.0,ORI_TYP #VAR,CIRC_TYP #BASE,JERK_FAC 50.0}
DECL FDAT FP466={TOOL_NO 0,BASE_NO 0,IPO_FRAME #BASE,POINT2[] " ",TQ_STATE FALSE}
DECL E6POS XP466={X 6109.20944,Y -705.3695,Z 3654.40552,A -102.70779,B 7.77597,C 4.76025,S 2,T 35,E1 -4140.9372,E2 0,E3 0,E4 0,E5 0,E6 0}
; DECL LDAT LCPDATP121={VEL 1,ACC 100,APO_DIST 100,APO_FAC 50.0,ORI_TYP #VAR,CIRC_TYP #BASE,JERK_FAC 50.0}
DECL FDAT FP467={TOOL_NO 0,BASE_NO 0,IPO_FRAME #BASE,POINT2[] " ",TQ_STATE FALSE}
DECL E6POS XP467={X 12777.06723,Y -602.17839,Z 3573.69413,A -83.4604,B -12.81532,C -0.94267,S 2,T 35,E1 -10812.08896,E2 0,E3 0,E4 0,E5 0,E6 0}
; DECL LDAT LCPDATP122={VEL 1,ACC 100,APO_DIST 100,APO_FAC 50.0,ORI_TYP #VAR,CIRC_TYP #BASE,JERK_FAC 50.0}
DECL FDAT FP468={TOOL_NO 0,BASE_NO 0,IPO_FRAME #BASE,POINT2[] " ",TQ_STATE FALSE}
DECL E6POS XP468={X 12675.92788,Y -569.18264,Z 3775.2407,A -83.4604,B -12.81532,C -0.94267,S 2,T 35,E1 -10812.08896,E2 0,E3 0,E4 0,E5 0,E6 0}
; DECL LDAT LCPDATP119={VEL 1,ACC 100,APO_DIST 100,APO_FAC 50.0,ORI_TYP #VAR,CIRC_TYP #BASE,JERK_FAC 50.0}
DECL FDAT FP469={TOOL_NO 0,BASE_NO 0,IPO_FRAME #BASE,POINT2[] " ",TQ_STATE FALSE}
DECL E6POS XP469={X 6034.81499,Y -708.12179,Z 3847.76366,A -102.7078,B 7.77596,C 4.76026,S 2,T 35,E1 -4174.36752,E2 0,E3 0,E4 0,E5 0,E6 0}
; DECL LDAT LCPDATP120={VEL 1,ACC 100,APO_DIST 100,APO_FAC 50.0,ORI_TYP #VAR,CIRC_TYP #BASE,JERK_FAC 50.0}
DECL FDAT FP470={TOOL_NO 0,BASE_NO 0,IPO_FRAME #BASE,POINT2[] " ",TQ_STATE FALSE}
DECL E6POS XP470={X 5808.56571,Y -717.10091,Z 4003.7046,A -102.70779,B 7.77596,C 4.76025,S 2,T 35,E1 -4005.10214,E2 0,E3 0,E4 0,E5 0,E6 0}
; DECL LDAT LCPDATP123={VEL 1,ACC 100,APO_DIST 100,APO_FAC 50.0,ORI_TYP #VAR,CIRC_TYP #BASE,JERK_FAC 50.0}
DECL FDAT FP471={TOOL_NO 0,BASE_NO 0,IPO_FRAME #BASE,POINT2[] " ",TQ_STATE FALSE}
DECL E6POS XP471={X 12607.03936,Y -538.48386,Z 3940.5062,A -83.4604,B -12.81532,C -0.94267,S 2,T 35,E1 -10812.08896,E2 0,E3 0,E4 0,E5 0,E6 0}
; DECL LDAT LCPDATP124={VEL 1,ACC 100,APO_DIST 100,APO_FAC 50.0,ORI_TYP #VAR,CIRC_TYP #BASE,JERK_FAC 50.0}
DECL FDAT FP472={TOOL_NO 0,BASE_NO 0,IPO_FRAME #BASE,POINT2[] " ",TQ_STATE FALSE}
DECL E6POS XP472={X 12329.73693,Y -538.48386,Z 3940.5062,A -83.38777,B -15.32829,C -1.2413,S 2,T 35,E1 -10812.08896,E2 0,E3 0,E4 0,E5 0,E6 0}
; DECL LDAT LCPDATP130={VEL 1,ACC 100,APO_DIST 100,APO_FAC 50.0,ORI_TYP #VAR,CIRC_TYP #BASE,JERK_FAC 50.0}
DECL FDAT FP473={TOOL_NO 0,BASE_NO 0,IPO_FRAME #BASE,POINT2[] " ",TQ_STATE FALSE}
DECL E6POS XP473={X 6035.27715,Y -717.10158,Z 4003.70466,A -106.51042,B 6.34838,C 5.00917,S 2,T 35,E1 -4231.81368,E2 0,E3 0,E4 0,E5 0,E6 0}
; DECL LDAT LCPDATP131={VEL 1,ACC 100,APO_DIST 100,APO_FAC 50.0,ORI_TYP #VAR,CIRC_TYP #BASE,JERK_FAC 50.0}
DECL FDAT FP474={TOOL_NO 0,BASE_NO 0,IPO_FRAME #BASE,POINT2[] " ",TQ_STATE FALSE}
DECL E6POS XP474={X 6001.84737,Y -717.10113,Z 4003.70421,A -106.4599,B 4.5615,C 5.54032,S 2,T 35,E1 -4198.38336,E2 0,E3 0,E4 0,E5 0,E6 0}
; DECL LDAT LCPDATP125={VEL 1,ACC 100,APO_DIST 100,APO_FAC 50.0,ORI_TYP #VAR,CIRC_TYP #BASE,JERK_FAC 50.0}
DECL FDAT FP475={TOOL_NO 0,BASE_NO 0,IPO_FRAME #BASE,POINT2[] " ",TQ_STATE FALSE}
DECL E6POS XP475={X 12327.62864,Y -538.48366,Z 3940.50597,A -87.76623,B -17.49847,C -1.50503,S 2,T 35,E1 -10473.34117,E2 0,E3 0,E4 0,E5 0,E6 0}
; DECL LDAT LCPDATP126={VEL 1,ACC 100,APO_DIST 100,APO_FAC 50.0,ORI_TYP #VAR,CIRC_TYP #BASE,JERK_FAC 50.0}
DECL FDAT FP476={TOOL_NO 0,BASE_NO 0,IPO_FRAME #BASE,POINT2[] " ",TQ_STATE FALSE}
DECL E6POS XP476={X 12344.44126,Y -538.48354,Z 3940.50612,A -92.12133,B -19.55447,C -1.59012,S 2,T 35,E1 -10490.15446,E2 0,E3 0,E4 0,E5 0,E6 0}
; DECL LDAT LCPDATP132={VEL 1,ACC 100,APO_DIST 100,APO_FAC 50.0,ORI_TYP #VAR,CIRC_TYP #BASE,JERK_FAC 50.0}
DECL FDAT FP477={TOOL_NO 0,BASE_NO 0,IPO_FRAME #BASE,POINT2[] " ",TQ_STATE FALSE}
DECL E6POS XP477={X 5984.60315,Y -717.10142,Z 4003.7045,A -107.27293,B 2.66443,C 6.10126,S 2,T 35,E1 -4181.13976,E2 0,E3 0,E4 0,E5 0,E6 0}
; DECL LDAT LCPDATP133={VEL 1,ACC 100,APO_DIST 100,APO_FAC 50.0,ORI_TYP #VAR,CIRC_TYP #BASE,JERK_FAC 50.0}
DECL FDAT FP478={TOOL_NO 0,BASE_NO 0,IPO_FRAME #BASE,POINT2[] " ",TQ_STATE FALSE}
DECL E6POS XP478={X 5959.53065,Y -717.10165,Z 4003.70439,A -107.25516,B 0.74219,C 6.69889,S 2,T 35,E1 -4156.06702,E2 0,E3 0,E4 0,E5 0,E6 0}
; DECL LDAT LCPDATP127={VEL 1,ACC 100,APO_DIST 100,APO_FAC 50.0,ORI_TYP #VAR,CIRC_TYP #BASE,JERK_FAC 50.0}
DECL FDAT FP479={TOOL_NO 0,BASE_NO 0,IPO_FRAME #BASE,POINT2[] " ",TQ_STATE FALSE}
DECL E6POS XP479={X 12327.65948,Y -538.48376,Z 3940.50627,A -96.02004,B -21.56802,C -1.50992,S 2,T 35,E1 -10473.37259,E2 0,E3 0,E4 0,E5 0,E6 0}
; DECL LDAT LCPDATP128={VEL 1,ACC 100,APO_DIST 100,APO_FAC 50.0,ORI_TYP #VAR,CIRC_TYP #BASE,JERK_FAC 50.0}
DECL FDAT FP480={TOOL_NO 0,BASE_NO 0,IPO_FRAME #BASE,POINT2[] " ",TQ_STATE FALSE}
DECL E6POS XP480={X 12434.40962,Y -538.48361,Z 3791.38491,A -100.48203,B -23.59142,C -1.27711,S 2,T 35,E1 -10580.12251,E2 0,E3 0,E4 0,E5 0,E6 0}
; DECL LDAT LCPDATP134={VEL 1,ACC 100,APO_DIST 100,APO_FAC 50.0,ORI_TYP #VAR,CIRC_TYP #BASE,JERK_FAC 50.0}
DECL FDAT FP481={TOOL_NO 0,BASE_NO 0,IPO_FRAME #BASE,POINT2[] " ",TQ_STATE FALSE}
DECL E6POS XP481={X 6027.18413,Y -717.10157,Z 4003.70451,A -108.83879,B -1.2655,C 7.3225,S 2,T 35,E1 -4223.72032,E2 0,E3 0,E4 0,E5 0,E6 0}
; DECL LDAT LCPDATP135={VEL 1,ACC 100,APO_DIST 100,APO_FAC 50.0,ORI_TYP #VAR,CIRC_TYP #BASE,JERK_FAC 50.0}
DECL FDAT FP482={TOOL_NO 0,BASE_NO 0,IPO_FRAME #BASE,POINT2[] " ",TQ_STATE FALSE}
DECL E6POS XP482={X 5994.01853,Y -717.10159,Z 4003.70409,A -109.42003,B -3.44272,C 8.06654,S 2,T 35,E1 -4190.55423,E2 0,E3 0,E4 0,E5 0,E6 0}
; DECL LDAT LCPDATP129={VEL 1,ACC 100,APO_DIST 100,APO_FAC 50.0,ORI_TYP #VAR,CIRC_TYP #BASE,JERK_FAC 50.0}
DECL FDAT FP483={TOOL_NO 0,BASE_NO 0,IPO_FRAME #BASE,POINT2[] " ",TQ_STATE FALSE}
DECL E6POS XP483={X 12525.53957,Y -538.48385,Z 3733.39322,A -103.74147,B -24.12805,C -1.24549,S 2,T 35,E1 -10671.25219,E2 0,E3 0,E4 0,E5 0,E6 0}
; DECL LDAT LCPDATP138={VEL 1,ACC 100,APO_DIST 100,APO_FAC 50.0,ORI_TYP #VAR,CIRC_TYP #BASE,JERK_FAC 50.0}
DECL FDAT FP484={TOOL_NO 0,BASE_NO 0,IPO_FRAME #BASE,POINT2[] " ",TQ_STATE FALSE}
DECL E6POS XP484={X 12409.55634,Y -538.48385,Z 3733.39322,A -103.74147,B -24.12805,C -1.24549,S 2,T 35,E1 -10555.26896,E2 0,E3 0,E4 0,E5 0,E6 0}
; DECL LDAT LCPDATP136={VEL 1,ACC 100,APO_DIST 100,APO_FAC 50.0,ORI_TYP #VAR,CIRC_TYP #BASE,JERK_FAC 50.0}
DECL FDAT FP485={TOOL_NO 0,BASE_NO 0,IPO_FRAME #BASE,POINT2[] " ",TQ_STATE FALSE}
DECL E6POS XP485={X 5960.30101,Y -717.10136,Z 4003.70387,A -109.95564,B -5.51238,C 8.79955,S 2,T 35,E1 -4156.83652,E2 0,E3 0,E4 0,E5 0,E6 0}
; DECL LDAT LCPDATP137={VEL 1,ACC 100,APO_DIST 100,APO_FAC 50.0,ORI_TYP #VAR,CIRC_TYP #BASE,JERK_FAC 50.0}
DECL FDAT FP486={TOOL_NO 0,BASE_NO 0,IPO_FRAME #BASE,POINT2[] " ",TQ_STATE FALSE}
DECL E6POS XP486={X 5959.29294,Y -717.10098,Z 4003.70454,A -110.58224,B -7.77816,C 9.62993,S 2,T 35,E1 -4155.82897,E2 0,E3 0,E4 0,E5 0,E6 0}
; DECL LDAT LCPDATP139={VEL 1,ACC 100,APO_DIST 100,APO_FAC 50.0,ORI_TYP #VAR,CIRC_TYP #BASE,JERK_FAC 50.0}
DECL FDAT FP487={TOOL_NO 0,BASE_NO 0,IPO_FRAME #BASE,POINT2[] " ",TQ_STATE FALSE}
DECL E6POS XP487={X 12666.37592,Y -538.48386,Z 3733.39329,A -110.95703,B -23.34196,C -1.63568,S 2,T 35,E1 -10812.08896,E2 0,E3 0,E4 0,E5 0,E6 0}
; DECL LDAT LCPDATP140={VEL 1,ACC 100,APO_DIST 100,APO_FAC 50.0,ORI_TYP #VAR,CIRC_TYP #BASE,JERK_FAC 50.0}
DECL FDAT FP488={TOOL_NO 0,BASE_NO 0,IPO_FRAME #BASE,POINT2[] " ",TQ_STATE FALSE}
DECL E6POS XP488={X 12666.37592,Y -538.48386,Z 3700.25522,A -113.36831,B -23.34196,C -1.63568,S 2,T 35,E1 -10812.08896,E2 0,E3 0,E4 0,E5 0,E6 0}
; DECL LDAT LCPDATP149={VEL 1,ACC 100,APO_DIST 100,APO_FAC 50.0,ORI_TYP #VAR,CIRC_TYP #BASE,JERK_FAC 50.0}
DECL FDAT FP489={TOOL_NO 0,BASE_NO 0,IPO_FRAME #BASE,POINT2[] " ",TQ_STATE FALSE}
DECL E6POS XP489={X 5916.8006,Y -717.10155,Z 4003.70412,A -110.72224,B -10.13455,C 10.52896,S 2,T 35,E1 -4113.33656,E2 0,E3 0,E4 0,E5 0,E6 0}
; DECL LDAT LCPDATP150={VEL 1,ACC 100,APO_DIST 100,APO_FAC 50.0,ORI_TYP #VAR,CIRC_TYP #BASE,JERK_FAC 50.0}
DECL FDAT FP490={TOOL_NO 0,BASE_NO 0,IPO_FRAME #BASE,POINT2[] " ",TQ_STATE FALSE}
DECL E6POS XP490={X 5875.31565,Y -717.1012,Z 4003.70448,A -110.8879,B -12.32973,C 11.37928,S 2,T 35,E1 -4071.85169,E2 0,E3 0,E4 0,E5 0,E6 0}
; DECL LDAT LCPDATP141={VEL 1,ACC 100,APO_DIST 100,APO_FAC 50.0,ORI_TYP #VAR,CIRC_TYP #BASE,JERK_FAC 50.0}
DECL FDAT FP491={TOOL_NO 0,BASE_NO 0,IPO_FRAME #BASE,POINT2[] " ",TQ_STATE FALSE}
DECL E6POS XP491={X 12666.37592,Y -538.48386,Z 3675.40167,A -115.34787,B -23.34196,C -1.63568,S 2,T 35,E1 -10812.08896,E2 0,E3 0,E4 0,E5 0,E6 0}
; DECL LDAT LCPDATP142={VEL 1,ACC 100,APO_DIST 100,APO_FAC 50.0,ORI_TYP #VAR,CIRC_TYP #BASE,JERK_FAC 50.0}
DECL FDAT FP492={TOOL_NO 0,BASE_NO 0,IPO_FRAME #BASE,POINT2[] " ",TQ_STATE FALSE}
DECL E6POS XP492={X 12666.37592,Y -538.48386,Z 3725.10877,A -117.62399,B -22.31862,C -2.21953,S 2,T 35,E1 -10812.08896,E2 0,E3 0,E4 0,E5 0,E6 0}
; DECL LDAT LCPDATP151={VEL 1,ACC 100,APO_DIST 100,APO_FAC 50.0,ORI_TYP #VAR,CIRC_TYP #BASE,JERK_FAC 50.0}
DECL FDAT FP493={TOOL_NO 0,BASE_NO 0,IPO_FRAME #BASE,POINT2[] " ",TQ_STATE FALSE}
DECL E6POS XP493={X 5898.57722,Y -717.10122,Z 4003.70435,A -112.09203,B -14.38754,C 12.19033,S 2,T 35,E1 -4095.11298,E2 0,E3 0,E4 0,E5 0,E6 0}
; DECL LDAT LCPDATP152={VEL 1,ACC 100,APO_DIST 100,APO_FAC 50.0,ORI_TYP #VAR,CIRC_TYP #BASE,JERK_FAC 50.0}
DECL FDAT FP494={TOOL_NO 0,BASE_NO 0,IPO_FRAME #BASE,POINT2[] " ",TQ_STATE FALSE}
DECL E6POS XP494={X 5854.40488,Y -717.10171,Z 4003.70448,A -112.35649,B -16.71303,C 13.17652,S 2,T 35,E1 -4050.94133,E2 0,E3 0,E4 0,E5 0,E6 0}
; DECL LDAT LCPDATP143={VEL 1,ACC 100,APO_DIST 100,APO_FAC 50.0,ORI_TYP #VAR,CIRC_TYP #BASE,JERK_FAC 50.0}
DECL FDAT FP495={TOOL_NO 0,BASE_NO 0,IPO_FRAME #BASE,POINT2[] " ",TQ_STATE FALSE}
DECL E6POS XP495={X 12666.37592,Y -538.48386,Z 3708.53974,A -119.39266,B -22.0406,C -2.38888,S 2,T 35,E1 -10812.08896,E2 0,E3 0,E4 0,E5 0,E6 0}
; DECL LDAT LCPDATP144={VEL 1,ACC 100,APO_DIST 100,APO_FAC 50.0,ORI_TYP #VAR,CIRC_TYP #BASE,JERK_FAC 50.0}
DECL FDAT FP496={TOOL_NO 0,BASE_NO 0,IPO_FRAME #BASE,POINT2[] " ",TQ_STATE FALSE}
DECL E6POS XP496={X 12666.37592,Y -538.48386,Z 3716.82426,A -121.52366,B -21.70131,C -2.61349,S 2,T 35,E1 -10812.08896,E2 0,E3 0,E4 0,E5 0,E6 0}
; DECL LDAT LCPDATP153={VEL 1,ACC 100,APO_DIST 100,APO_FAC 50.0,ORI_TYP #VAR,CIRC_TYP #BASE,JERK_FAC 50.0}
DECL FDAT FP497={TOOL_NO 0,BASE_NO 0,IPO_FRAME #BASE,POINT2[] " ",TQ_STATE FALSE}
DECL E6POS XP497={X 5865.70091,Y -717.10124,Z 4003.70383,A -113.62634,B -18.80667,C 14.08679,S 2,T 35,E1 -4062.23613,E2 0,E3 0,E4 0,E5 0,E6 0}
; DECL LDAT LCPDATP154={VEL 1,ACC 100,APO_DIST 100,APO_FAC 50.0,ORI_TYP #VAR,CIRC_TYP #BASE,JERK_FAC 50.0}
DECL FDAT FP498={TOOL_NO 0,BASE_NO 0,IPO_FRAME #BASE,POINT2[] " ",TQ_STATE FALSE}
DECL E6POS XP498={X 5786.97193,Y -717.10138,Z 4003.70442,A -113.90846,B -20.59534,C 14.92344,S 2,T 35,E1 -3983.50839,E2 0,E3 0,E4 0,E5 0,E6 0}
; DECL LDAT LCPDATP145={VEL 1,ACC 100,APO_DIST 100,APO_FAC 50.0,ORI_TYP #VAR,CIRC_TYP #BASE,JERK_FAC 50.0}
DECL FDAT FP499={TOOL_NO 0,BASE_NO 0,IPO_FRAME #BASE,POINT2[] " ",TQ_STATE FALSE}
DECL E6POS XP499={X 12666.37592,Y -538.48386,Z 3691.97071,A -122.58569,B -21.70131,C -2.61349,S 2,T 35,E1 -10812.08896,E2 0,E3 0,E4 0,E5 0,E6 0}
; DECL LDAT LCPDATP146={VEL 1,ACC 100,APO_DIST 100,APO_FAC 50.0,ORI_TYP #VAR,CIRC_TYP #BASE,JERK_FAC 50.0}
DECL FDAT FP500={TOOL_NO 0,BASE_NO 0,IPO_FRAME #BASE,POINT2[] " ",TQ_STATE FALSE}
DECL E6POS XP500={X 12666.37592,Y -538.48386,Z 3741.67781,A -124.88801,B -20.60151,C -3.44033,S 2,T 35,E1 -10812.08896,E2 0,E3 0,E4 0,E5 0,E6 0}
; DECL LDAT LCPDATP155={VEL 1,ACC 100,APO_DIST 100,APO_FAC 50.0,ORI_TYP #VAR,CIRC_TYP #BASE,JERK_FAC 50.0}
DECL FDAT FP501={TOOL_NO 0,BASE_NO 0,IPO_FRAME #BASE,POINT2[] " ",TQ_STATE FALSE}
DECL E6POS XP501={X 5766.06143,Y -717.10078,Z 4003.7047,A -114.88478,B -21.82725,C 15.51221,S 2,T 35,E1 -3962.59803,E2 0,E3 0,E4 0,E5 0,E6 0}
; DECL LDAT LCPDATP156={VEL 1,ACC 100,APO_DIST 100,APO_FAC 50.0,ORI_TYP #VAR,CIRC_TYP #BASE,JERK_FAC 50.0}
DECL FDAT FP502={TOOL_NO 0,BASE_NO 0,IPO_FRAME #BASE,POINT2[] " ",TQ_STATE FALSE}
DECL E6POS XP502={X 5671.46198,Y -717.1018,Z 4003.704,A -116.65787,B -23.21109,C 16.21129,S 2,T 35,E1 -3867.99764,E2 0,E3 0,E4 0,E5 0,E6 0}
; DECL LDAT LCPDATP147={VEL 1,ACC 100,APO_DIST 100,APO_FAC 50.0,ORI_TYP #VAR,CIRC_TYP #BASE,JERK_FAC 50.0}
DECL FDAT FP503={TOOL_NO 0,BASE_NO 0,IPO_FRAME #BASE,POINT2[] " ",TQ_STATE FALSE}
DECL E6POS XP503={X 12666.37592,Y -538.48386,Z 3708.53974,A -127.07895,B -20.60151,C -3.44033,S 2,T 35,E1 -10812.08896,E2 0,E3 0,E4 0,E5 0,E6 0}
; DECL LDAT LCPDATP113={VEL 1,ACC 100,APO_DIST 100,APO_FAC 50.0,ORI_TYP #VAR,CIRC_TYP #BASE,JERK_FAC 50.0}
DECL FDAT FP504={TOOL_NO 0,BASE_NO 0,IPO_FRAME #BASE,POINT2[] " ",TQ_STATE FALSE}
DECL E6POS XP504={X 6379.94734,Y -681.40788,Z 3158.20554,A -102.40256,B 11.37187,C 4.81103,S 2,T 35,E1 -4209.91162,E2 0,E3 0,E4 0,E5 0,E6 0}
; DECL LDAT LCPDATP114={VEL 1,ACC 100,APO_DIST 100,APO_FAC 50.0,ORI_TYP #VAR,CIRC_TYP #BASE,JERK_FAC 50.0}
DECL FDAT FP505={TOOL_NO 0,BASE_NO 0,IPO_FRAME #BASE,POINT2[] " ",TQ_STATE FALSE}
DECL E6POS XP505={X 6328.481,Y -681.40737,Z 3158.20597,A -102.7078,B 7.77597,C 4.76025,S 2,T 35,E1 -4158.44503,E2 0,E3 0,E4 0,E5 0,E6 0}
; DECL LDAT LCPDATP115={VEL 1,ACC 100,APO_DIST 100,APO_FAC 50.0,ORI_TYP #VAR,CIRC_TYP #BASE,JERK_FAC 50.0}
DECL FDAT FP506={TOOL_NO 0,BASE_NO 0,IPO_FRAME #BASE,POINT2[] " ",TQ_STATE FALSE}
DECL E6POS XP506={X 12929.38089,Y -681.40737,Z 3158.20639,A -83.4604,B -12.81532,C -0.94267,S 2,T 35,E1 -10812.08896,E2 0,E3 0,E4 0,E5 0,E6 0}
; DECL LDAT LCPDATP116={VEL 1,ACC 100,APO_DIST 100,APO_FAC 50.0,ORI_TYP #VAR,CIRC_TYP #BASE,JERK_FAC 50.0}
DECL FDAT FP507={TOOL_NO 0,BASE_NO 0,IPO_FRAME #BASE,POINT2[] " ",TQ_STATE FALSE}
DECL E6POS XP507={X 12886.08572,Y -646.4113,Z 3336.02814,A -83.4604,B -12.81532,C -0.94267,S 2,T 35,E1 -10812.08896,E2 0,E3 0,E4 0,E5 0,E6 0}
; DECL LDAT LCPDATP117={VEL 1,ACC 100,APO_DIST 100,APO_FAC 50.0,ORI_TYP #VAR,CIRC_TYP #BASE,JERK_FAC 50.0}
DECL FDAT FP508={TOOL_NO 0,BASE_NO 0,IPO_FRAME #BASE,POINT2[] " ",TQ_STATE FALSE}
DECL E6POS XP508={X 6226.20694,Y -691.76303,Z 3410.82553,A -102.7078,B 7.77597,C 4.76022,S 2,T 35,E1 -4167.06683,E2 0,E3 0,E4 0,E5 0,E6 0}
; DECL LDAT LCPDATP118={VEL 1,ACC 100,APO_DIST 100,APO_FAC 50.0,ORI_TYP #VAR,CIRC_TYP #BASE,JERK_FAC 50.0}
DECL FDAT FP509={TOOL_NO 0,BASE_NO 0,IPO_FRAME #BASE,POINT2[] " ",TQ_STATE FALSE}
DECL E6POS XP509={X 6109.20944,Y -705.3695,Z 3654.40552,A -102.70779,B 7.77597,C 4.76025,S 2,T 35,E1 -4140.9372,E2 0,E3 0,E4 0,E5 0,E6 0}
; DECL LDAT LCPDATP121={VEL 1,ACC 100,APO_DIST 100,APO_FAC 50.0,ORI_TYP #VAR,CIRC_TYP #BASE,JERK_FAC 50.0}
DECL FDAT FP510={TOOL_NO 0,BASE_NO 0,IPO_FRAME #BASE,POINT2[] " ",TQ_STATE FALSE}
DECL E6POS XP510={X 12777.06723,Y -602.17839,Z 3573.69413,A -83.4604,B -12.81532,C -0.94267,S 2,T 35,E1 -10812.08896,E2 0,E3 0,E4 0,E5 0,E6 0}
; DECL LDAT LCPDATP122={VEL 1,ACC 100,APO_DIST 100,APO_FAC 50.0,ORI_TYP #VAR,CIRC_TYP #BASE,JERK_FAC 50.0}
DECL FDAT FP511={TOOL_NO 0,BASE_NO 0,IPO_FRAME #BASE,POINT2[] " ",TQ_STATE FALSE}
DECL E6POS XP511={X 12675.92788,Y -569.18264,Z 3775.2407,A -83.4604,B -12.81532,C -0.94267,S 2,T 35,E1 -10812.08896,E2 0,E3 0,E4 0,E5 0,E6 0}
; DECL LDAT LCPDATP119={VEL 1,ACC 100,APO_DIST 100,APO_FAC 50.0,ORI_TYP #VAR,CIRC_TYP #BASE,JERK_FAC 50.0}
DECL FDAT FP512={TOOL_NO 0,BASE_NO 0,IPO_FRAME #BASE,POINT2[] " ",TQ_STATE FALSE}
DECL E6POS XP512={X 6034.81499,Y -708.12179,Z 3847.76366,A -102.7078,B 7.77596,C 4.76026,S 2,T 35,E1 -4174.36752,E2 0,E3 0,E4 0,E5 0,E6 0}
; DECL LDAT LCPDATP120={VEL 1,ACC 100,APO_DIST 100,APO_FAC 50.0,ORI_TYP #VAR,CIRC_TYP #BASE,JERK_FAC 50.0}
DECL FDAT FP513={TOOL_NO 0,BASE_NO 0,IPO_FRAME #BASE,POINT2[] " ",TQ_STATE FALSE}
DECL E6POS XP513={X 5808.56571,Y -717.10091,Z 4003.7046,A -102.70779,B 7.77596,C 4.76025,S 2,T 35,E1 -4005.10214,E2 0,E3 0,E4 0,E5 0,E6 0}
; DECL LDAT LCPDATP123={VEL 1,ACC 100,APO_DIST 100,APO_FAC 50.0,ORI_TYP #VAR,CIRC_TYP #BASE,JERK_FAC 50.0}
DECL FDAT FP514={TOOL_NO 0,BASE_NO 0,IPO_FRAME #BASE,POINT2[] " ",TQ_STATE FALSE}
DECL E6POS XP514={X 12607.03936,Y -538.48386,Z 3940.5062,A -83.4604,B -12.81532,C -0.94267,S 2,T 35,E1 -10812.08896,E2 0,E3 0,E4 0,E5 0,E6 0}
; DECL LDAT LCPDATP124={VEL 1,ACC 100,APO_DIST 100,APO_FAC 50.0,ORI_TYP #VAR,CIRC_TYP #BASE,JERK_FAC 50.0}
DECL FDAT FP515={TOOL_NO 0,BASE_NO 0,IPO_FRAME #BASE,POINT2[] " ",TQ_STATE FALSE}
DECL E6POS XP515={X 12329.73693,Y -538.48386,Z 3940.5062,A -83.38777,B -15.32829,C -1.2413,S 2,T 35,E1 -10812.08896,E2 0,E3 0,E4 0,E5 0,E6 0}
; DECL LDAT LCPDATP130={VEL 1,ACC 100,APO_DIST 100,APO_FAC 50.0,ORI_TYP #VAR,CIRC_TYP #BASE,JERK_FAC 50.0}
DECL FDAT FP516={TOOL_NO 0,BASE_NO 0,IPO_FRAME #BASE,POINT2[] " ",TQ_STATE FALSE}
DECL E6POS XP516={X 6035.27715,Y -717.10158,Z 4003.70466,A -106.51042,B 6.34838,C 5.00917,S 2,T 35,E1 -4231.81368,E2 0,E3 0,E4 0,E5 0,E6 0}
; DECL LDAT LCPDATP131={VEL 1,ACC 100,APO_DIST 100,APO_FAC 50.0,ORI_TYP #VAR,CIRC_TYP #BASE,JERK_FAC 50.0}
DECL FDAT FP517={TOOL_NO 0,BASE_NO 0,IPO_FRAME #BASE,POINT2[] " ",TQ_STATE FALSE}
DECL E6POS XP517={X 6001.84737,Y -717.10113,Z 4003.70421,A -106.4599,B 4.5615,C 5.54032,S 2,T 35,E1 -4198.38336,E2 0,E3 0,E4 0,E5 0,E6 0}
; DECL LDAT LCPDATP125={VEL 1,ACC 100,APO_DIST 100,APO_FAC 50.0,ORI_TYP #VAR,CIRC_TYP #BASE,JERK_FAC 50.0}
DECL FDAT FP518={TOOL_NO 0,BASE_NO 0,IPO_FRAME #BASE,POINT2[] " ",TQ_STATE FALSE}
DECL E6POS XP518={X 12327.62864,Y -538.48366,Z 3940.50597,A -87.76623,B -17.49847,C -1.50503,S 2,T 35,E1 -10473.34117,E2 0,E3 0,E4 0,E5 0,E6 0}
; DECL LDAT LCPDATP126={VEL 1,ACC 100,APO_DIST 100,APO_FAC 50.0,ORI_TYP #VAR,CIRC_TYP #BASE,JERK_FAC 50.0}
DECL FDAT FP519={TOOL_NO 0,BASE_NO 0,IPO_FRAME #BASE,POINT2[] " ",TQ_STATE FALSE}
DECL E6POS XP519={X 12344.44126,Y -538.48354,Z 3940.50612,A -92.12133,B -19.55447,C -1.59012,S 2,T 35,E1 -10490.15446,E2 0,E3 0,E4 0,E5 0,E6 0}
; DECL LDAT LCPDATP132={VEL 1,ACC 100,APO_DIST 100,APO_FAC 50.0,ORI_TYP #VAR,CIRC_TYP #BASE,JERK_FAC 50.0}
DECL FDAT FP520={TOOL_NO 0,BASE_NO 0,IPO_FRAME #BASE,POINT2[] " ",TQ_STATE FALSE}
DECL E6POS XP520={X 5984.60315,Y -717.10142,Z 4003.7045,A -107.27293,B 2.66443,C 6.10126,S 2,T 35,E1 -4181.13976,E2 0,E3 0,E4 0,E5 0,E6 0}
; DECL LDAT LCPDATP133={VEL 1,ACC 100,APO_DIST 100,APO_FAC 50.0,ORI_TYP #VAR,CIRC_TYP #BASE,JERK_FAC 50.0}
DECL FDAT FP521={TOOL_NO 0,BASE_NO 0,IPO_FRAME #BASE,POINT2[] " ",TQ_STATE FALSE}
DECL E6POS XP521={X 5959.53065,Y -717.10165,Z 4003.70439,A -107.25516,B 0.74219,C 6.69889,S 2,T 35,E1 -4156.06702,E2 0,E3 0,E4 0,E5 0,E6 0}
; DECL LDAT LCPDATP127={VEL 1,ACC 100,APO_DIST 100,APO_FAC 50.0,ORI_TYP #VAR,CIRC_TYP #BASE,JERK_FAC 50.0}
DECL FDAT FP522={TOOL_NO 0,BASE_NO 0,IPO_FRAME #BASE,POINT2[] " ",TQ_STATE FALSE}
DECL E6POS XP522={X 12327.65948,Y -538.48376,Z 3940.50627,A -96.02004,B -21.56802,C -1.50992,S 2,T 35,E1 -10473.37259,E2 0,E3 0,E4 0,E5 0,E6 0}
; DECL LDAT LCPDATP128={VEL 1,ACC 100,APO_DIST 100,APO_FAC 50.0,ORI_TYP #VAR,CIRC_TYP #BASE,JERK_FAC 50.0}
DECL FDAT FP523={TOOL_NO 0,BASE_NO 0,IPO_FRAME #BASE,POINT2[] " ",TQ_STATE FALSE}
DECL E6POS XP523={X 12434.40962,Y -538.48361,Z 3791.38491,A -100.48203,B -23.59142,C -1.27711,S 2,T 35,E1 -10580.12251,E2 0,E3 0,E4 0,E5 0,E6 0}
; DECL LDAT LCPDATP134={VEL 1,ACC 100,APO_DIST 100,APO_FAC 50.0,ORI_TYP #VAR,CIRC_TYP #BASE,JERK_FAC 50.0}
DECL FDAT FP524={TOOL_NO 0,BASE_NO 0,IPO_FRAME #BASE,POINT2[] " ",TQ_STATE FALSE}
DECL E6POS XP524={X 6027.18413,Y -717.10157,Z 4003.70451,A -108.83879,B -1.2655,C 7.3225,S 2,T 35,E1 -4223.72032,E2 0,E3 0,E4 0,E5 0,E6 0}
; DECL LDAT LCPDATP135={VEL 1,ACC 100,APO_DIST 100,APO_FAC 50.0,ORI_TYP #VAR,CIRC_TYP #BASE,JERK_FAC 50.0}
DECL FDAT FP525={TOOL_NO 0,BASE_NO 0,IPO_FRAME #BASE,POINT2[] " ",TQ_STATE FALSE}
DECL E6POS XP525={X 5994.01853,Y -717.10159,Z 4003.70409,A -109.42003,B -3.44272,C 8.06654,S 2,T 35,E1 -4190.55423,E2 0,E3 0,E4 0,E5 0,E6 0}
; DECL LDAT LCPDATP129={VEL 1,ACC 100,APO_DIST 100,APO_FAC 50.0,ORI_TYP #VAR,CIRC_TYP #BASE,JERK_FAC 50.0}
DECL FDAT FP526={TOOL_NO 0,BASE_NO 0,IPO_FRAME #BASE,POINT2[] " ",TQ_STATE FALSE}
DECL E6POS XP526={X 12525.53957,Y -538.48385,Z 3733.39322,A -103.74147,B -24.12805,C -1.24549,S 2,T 35,E1 -10671.25219,E2 0,E3 0,E4 0,E5 0,E6 0}
; DECL LDAT LCPDATP138={VEL 1,ACC 100,APO_DIST 100,APO_FAC 50.0,ORI_TYP #VAR,CIRC_TYP #BASE,JERK_FAC 50.0}
DECL FDAT FP527={TOOL_NO 0,BASE_NO 0,IPO_FRAME #BASE,POINT2[] " ",TQ_STATE FALSE}
DECL E6POS XP527={X 12409.55634,Y -538.48385,Z 3733.39322,A -103.74147,B -24.12805,C -1.24549,S 2,T 35,E1 -10555.26896,E2 0,E3 0,E4 0,E5 0,E6 0}
; DECL LDAT LCPDATP136={VEL 1,ACC 100,APO_DIST 100,APO_FAC 50.0,ORI_TYP #VAR,CIRC_TYP #BASE,JERK_FAC 50.0}
DECL FDAT FP528={TOOL_NO 0,BASE_NO 0,IPO_FRAME #BASE,POINT2[] " ",TQ_STATE FALSE}
DECL E6POS XP528={X 5960.30101,Y -717.10136,Z 4003.70387,A -109.95564,B -5.51238,C 8.79955,S 2,T 35,E1 -4156.83652,E2 0,E3 0,E4 0,E5 0,E6 0}
; DECL LDAT LCPDATP137={VEL 1,ACC 100,APO_DIST 100,APO_FAC 50.0,ORI_TYP #VAR,CIRC_TYP #BASE,JERK_FAC 50.0}
DECL FDAT FP529={TOOL_NO 0,BASE_NO 0,IPO_FRAME #BASE,POINT2[] " ",TQ_STATE FALSE}
DECL E6POS XP529={X 5959.29294,Y -717.10098,Z 4003.70454,A -110.58224,B -7.77816,C 9.62993,S 2,T 35,E1 -4155.82897,E2 0,E3 0,E4 0,E5 0,E6 0}
; DECL LDAT LCPDATP139={VEL 1,ACC 100,APO_DIST 100,APO_FAC 50.0,ORI_TYP #VAR,CIRC_TYP #BASE,JERK_FAC 50.0}
DECL FDAT FP530={TOOL_NO 0,BASE_NO 0,IPO_FRAME #BASE,POINT2[] " ",TQ_STATE FALSE}
DECL E6POS XP530={X 12666.37592,Y -538.48386,Z 3733.39329,A -110.95703,B -23.34196,C -1.63568,S 2,T 35,E1 -10812.08896,E2 0,E3 0,E4 0,E5 0,E6 0}
; DECL LDAT LCPDATP140={VEL 1,ACC 100,APO_DIST 100,APO_FAC 50.0,ORI_TYP #VAR,CIRC_TYP #BASE,JERK_FAC 50.0}
DECL FDAT FP531={TOOL_NO 0,BASE_NO 0,IPO_FRAME #BASE,POINT2[] " ",TQ_STATE FALSE}
DECL E6POS XP531={X 12666.37592,Y -538.48386,Z 3700.25522,A -113.36831,B -23.34196,C -1.63568,S 2,T 35,E1 -10812.08896,E2 0,E3 0,E4 0,E5 0,E6 0}
; DECL LDAT LCPDATP149={VEL 1,ACC 100,APO_DIST 100,APO_FAC 50.0,ORI_TYP #VAR,CIRC_TYP #BASE,JERK_FAC 50.0}
DECL FDAT FP532={TOOL_NO 0,BASE_NO 0,IPO_FRAME #BASE,POINT2[] " ",TQ_STATE FALSE}
DECL E6POS XP532={X 5916.8006,Y -717.10155,Z 4003.70412,A -110.72224,B -10.13455,C 10.52896,S 2,T 35,E1 -4113.33656,E2 0,E3 0,E4 0,E5 0,E6 0}
; DECL LDAT LCPDATP150={VEL 1,ACC 100,APO_DIST 100,APO_FAC 50.0,ORI_TYP #VAR,CIRC_TYP #BASE,JERK_FAC 50.0}
DECL FDAT FP533={TOOL_NO 0,BASE_NO 0,IPO_FRAME #BASE,POINT2[] " ",TQ_STATE FALSE}
DECL E6POS XP533={X 5875.31565,Y -717.1012,Z 4003.70448,A -110.8879,B -12.32973,C 11.37928,S 2,T 35,E1 -4071.85169,E2 0,E3 0,E4 0,E5 0,E6 0}
; DECL LDAT LCPDATP141={VEL 1,ACC 100,APO_DIST 100,APO_FAC 50.0,ORI_TYP #VAR,CIRC_TYP #BASE,JERK_FAC 50.0}
DECL FDAT FP534={TOOL_NO 0,BASE_NO 0,IPO_FRAME #BASE,POINT2[] " ",TQ_STATE FALSE}
DECL E6POS XP534={X 12666.37592,Y -538.48386,Z 3675.40167,A -115.34787,B -23.34196,C -1.63568,S 2,T 35,E1 -10812.08896,E2 0,E3 0,E4 0,E5 0,E6 0}
; DECL LDAT LCPDATP142={VEL 1,ACC 100,APO_DIST 100,APO_FAC 50.0,ORI_TYP #VAR,CIRC_TYP #BASE,JERK_FAC 50.0}
DECL FDAT FP535={TOOL_NO 0,BASE_NO 0,IPO_FRAME #BASE,POINT2[] " ",TQ_STATE FALSE}
DECL E6POS XP535={X 12666.37592,Y -538.48386,Z 3725.10877,A -117.62399,B -22.31862,C -2.21953,S 2,T 35,E1 -10812.08896,E2 0,E3 0,E4 0,E5 0,E6 0}
; DECL LDAT LCPDATP151={VEL 1,ACC 100,APO_DIST 100,APO_FAC 50.0,ORI_TYP #VAR,CIRC_TYP #BASE,JERK_FAC 50.0}
DECL FDAT FP536={TOOL_NO 0,BASE_NO 0,IPO_FRAME #BASE,POINT2[] " ",TQ_STATE FALSE}
DECL E6POS XP536={X 5898.57722,Y -717.10122,Z 4003.70435,A -112.09203,B -14.38754,C 12.19033,S 2,T 35,E1 -4095.11298,E2 0,E3 0,E4 0,E5 0,E6 0}
; DECL LDAT LCPDATP152={VEL 1,ACC 100,APO_DIST 100,APO_FAC 50.0,ORI_TYP #VAR,CIRC_TYP #BASE,JERK_FAC 50.0}
DECL FDAT FP537={TOOL_NO 0,BASE_NO 0,IPO_FRAME #BASE,POINT2[] " ",TQ_STATE FALSE}
DECL E6POS XP537={X 5854.40488,Y -717.10171,Z 4003.70448,A -112.35649,B -16.71303,C 13.17652,S 2,T 35,E1 -4050.94133,E2 0,E3 0,E4 0,E5 0,E6 0}
; DECL LDAT LCPDATP143={VEL 1,ACC 100,APO_DIST 100,APO_FAC 50.0,ORI_TYP #VAR,CIRC_TYP #BASE,JERK_FAC 50.0}
DECL FDAT FP538={TOOL_NO 0,BASE_NO 0,IPO_FRAME #BASE,POINT2[] " ",TQ_STATE FALSE}
DECL E6POS XP538={X 12666.37592,Y -538.48386,Z 3708.53974,A -119.39266,B -22.0406,C -2.38888,S 2,T 35,E1 -10812.08896,E2 0,E3 0,E4 0,E5 0,E6 0}
; DECL LDAT LCPDATP144={VEL 1,ACC 100,APO_DIST 100,APO_FAC 50.0,ORI_TYP #VAR,CIRC_TYP #BASE,JERK_FAC 50.0}
DECL FDAT FP539={TOOL_NO 0,BASE_NO 0,IPO_FRAME #BASE,POINT2[] " ",TQ_STATE FALSE}
DECL E6POS XP539={X 12666.37592,Y -538.48386,Z 3716.82426,A -121.52366,B -21.70131,C -2.61349,S 2,T 35,E1 -10812.08896,E2 0,E3 0,E4 0,E5 0,E6 0}
; DECL LDAT LCPDATP153={VEL 1,ACC 100,APO_DIST 100,APO_FAC 50.0,ORI_TYP #VAR,CIRC_TYP #BASE,JERK_FAC 50.0}
DECL FDAT FP540={TOOL_NO 0,BASE_NO 0,IPO_FRAME #BASE,POINT2[] " ",TQ_STATE FALSE}
DECL E6POS XP540={X 5865.70091,Y -717.10124,Z 4003.70383,A -113.62634,B -18.80667,C 14.08679,S 2,T 35,E1 -4062.23613,E2 0,E3 0,E4 0,E5 0,E6 0}
; DECL LDAT LCPDATP154={VEL 1,ACC 100,APO_DIST 100,APO_FAC 50.0,ORI_TYP #VAR,CIRC_TYP #BASE,JERK_FAC 50.0}
DECL FDAT FP541={TOOL_NO 0,BASE_NO 0,IPO_FRAME #BASE,POINT2[] " ",TQ_STATE FALSE}
DECL E6POS XP541={X 5786.97193,Y -717.10138,Z 4003.70442,A -113.90846,B -20.59534,C 14.92344,S 2,T 35,E1 -3983.50839,E2 0,E3 0,E4 0,E5 0,E6 0}
; DECL LDAT LCPDATP145={VEL 1,ACC 100,APO_DIST 100,APO_FAC 50.0,ORI_TYP #VAR,CIRC_TYP #BASE,JERK_FAC 50.0}
DECL FDAT FP542={TOOL_NO 0,BASE_NO 0,IPO_FRAME #BASE,POINT2[] " ",TQ_STATE FALSE}
DECL E6POS XP542={X 12666.37592,Y -538.48386,Z 3691.97071,A -122.58569,B -21.70131,C -2.61349,S 2,T 35,E1 -10812.08896,E2 0,E3 0,E4 0,E5 0,E6 0}
; DECL LDAT LCPDATP146={VEL 1,ACC 100,APO_DIST 100,APO_FAC 50.0,ORI_TYP #VAR,CIRC_TYP #BASE,JERK_FAC 50.0}
DECL FDAT FP543={TOOL_NO 0,BASE_NO 0,IPO_FRAME #BASE,POINT2[] " ",TQ_STATE FALSE}
DECL E6POS XP543={X 12666.37592,Y -538.48386,Z 3741.67781,A -124.88801,B -20.60151,C -3.44033,S 2,T 35,E1 -10812.08896,E2 0,E3 0,E4 0,E5 0,E6 0}
; DECL LDAT LCPDATP155={VEL 1,ACC 100,APO_DIST 100,APO_FAC 50.0,ORI_TYP #VAR,CIRC_TYP #BASE,JERK_FAC 50.0}
DECL FDAT FP544={TOOL_NO 0,BASE_NO 0,IPO_FRAME #BASE,POINT2[] " ",TQ_STATE FALSE}
DECL E6POS XP544={X 5766.06143,Y -717.10078,Z 4003.7047,A -114.88478,B -21.82725,C 15.51221,S 2,T 35,E1 -3962.59803,E2 0,E3 0,E4 0,E5 0,E6 0}
; DECL LDAT LCPDATP156={VEL 1,ACC 100,APO_DIST 100,APO_FAC 50.0,ORI_TYP #VAR,CIRC_TYP #BASE,JERK_FAC 50.0}
DECL FDAT FP545={TOOL_NO 0,BASE_NO 0,IPO_FRAME #BASE,POINT2[] " ",TQ_STATE FALSE}
DECL E6POS XP545={X 5671.46198,Y -717.1018,Z 4003.704,A -116.65787,B -23.21109,C 16.21129,S 2,T 35,E1 -3867.99764,E2 0,E3 0,E4 0,E5 0,E6 0}
; DECL LDAT LCPDATP147={VEL 1,ACC 100,APO_DIST 100,APO_FAC 50.0,ORI_TYP #VAR,CIRC_TYP #BASE,JERK_FAC 50.0}
DECL FDAT FP546={TOOL_NO 0,BASE_NO 0,IPO_FRAME #BASE,POINT2[] " ",TQ_STATE FALSE}
DECL E6POS XP546={X 12666.37592,Y -538.48386,Z 3708.53974,A -127.07895,B -20.60151,C -3.44033,S 2,T 35,E1 -10812.08896,E2 0,E3 0,E4 0,E5 0,E6 0}
; DECL LDAT LCPDATP113={VEL 1,ACC 100,APO_DIST 100,APO_FAC 50.0,ORI_TYP #VAR,CIRC_TYP #BASE,JERK_FAC 50.0}
DECL FDAT FP547={TOOL_NO 0,BASE_NO 0,IPO_FRAME #BASE,POINT2[] " ",TQ_STATE FALSE}
DECL E6POS XP547={X 6379.94734,Y -681.40788,Z 3158.20554,A -102.40256,B 11.37187,C 4.81103,S 2,T 35,E1 -4209.91162,E2 0,E3 0,E4 0,E5 0,E6 0}
; DECL LDAT LCPDATP114={VEL 1,ACC 100,APO_DIST 100,APO_FAC 50.0,ORI_TYP #VAR,CIRC_TYP #BASE,JERK_FAC 50.0}
DECL FDAT FP548={TOOL_NO 0,BASE_NO 0,IPO_FRAME #BASE,POINT2[] " ",TQ_STATE FALSE}
DECL E6POS XP548={X 6328.481,Y -681.40737,Z 3158.20597,A -102.7078,B 7.77597,C 4.76025,S 2,T 35,E1 -4158.44503,E2 0,E3 0,E4 0,E5 0,E6 0}
; DECL LDAT LCPDATP115={VEL 1,ACC 100,APO_DIST 100,APO_FAC 50.0,ORI_TYP #VAR,CIRC_TYP #BASE,JERK_FAC 50.0}
DECL FDAT FP549={TOOL_NO 0,BASE_NO 0,IPO_FRAME #BASE,POINT2[] " ",TQ_STATE FALSE}
DECL E6POS XP549={X 12929.38089,Y -681.40737,Z 3158.20639,A -83.4604,B -12.81532,C -0.94267,S 2,T 35,E1 -10812.08896,E2 0,E3 0,E4 0,E5 0,E6 0}
; DECL LDAT LCPDATP116={VEL 1,ACC 100,APO_DIST 100,APO_FAC 50.0,ORI_TYP #VAR,CIRC_TYP #BASE,JERK_FAC 50.0}
DECL FDAT FP550={TOOL_NO 0,BASE_NO 0,IPO_FRAME #BASE,POINT2[] " ",TQ_STATE FALSE}
DECL E6POS XP550={X 12886.08572,Y -646.4113,Z 3336.02814,A -83.4604,B -12.81532,C -0.94267,S 2,T 35,E1 -10812.08896,E2 0,E3 0,E4 0,E5 0,E6 0}
; DECL LDAT LCPDATP117={VEL 1,ACC 100,APO_DIST 100,APO_FAC 50.0,ORI_TYP #VAR,CIRC_TYP #BASE,JERK_FAC 50.0}
DECL FDAT FP551={TOOL_NO 0,BASE_NO 0,IPO_FRAME #BASE,POINT2[] " ",TQ_STATE FALSE}
DECL E6POS XP551={X 6226.20694,Y -691.76303,Z 3410.82553,A -102.7078,B 7.77597,C 4.76022,S 2,T 35,E1 -4167.06683,E2 0,E3 0,E4 0,E5 0,E6 0}
; DECL LDAT LCPDATP118={VEL 1,ACC 100,APO_DIST 100,APO_FAC 50.0,ORI_TYP #VAR,CIRC_TYP #BASE,JERK_FAC 50.0}
DECL FDAT FP552={TOOL_NO 0,BASE_NO 0,IPO_FRAME #BASE,POINT2[] " ",TQ_STATE FALSE}
DECL E6POS XP552={X 6109.20944,Y -705.3695,Z 3654.40552,A -102.70779,B 7.77597,C 4.76025,S 2,T 35,E1 -4140.9372,E2 0,E3 0,E4 0,E5 0,E6 0}
; DECL LDAT LCPDATP121={VEL 1,ACC 100,APO_DIST 100,APO_FAC 50.0,ORI_TYP #VAR,CIRC_TYP #BASE,JERK_FAC 50.0}
DECL FDAT FP553={TOOL_NO 0,BASE_NO 0,IPO_FRAME #BASE,POINT2[] " ",TQ_STATE FALSE}
DECL E6POS XP553={X 12777.06723,Y -602.17839,Z 3573.69413,A -83.4604,B -12.81532,C -0.94267,S 2,T 35,E1 -10812.08896,E2 0,E3 0,E4 0,E5 0,E6 0}
; DECL LDAT LCPDATP122={VEL 1,ACC 100,APO_DIST 100,APO_FAC 50.0,ORI_TYP #VAR,CIRC_TYP #BASE,JERK_FAC 50.0}
DECL FDAT FP554={TOOL_NO 0,BASE_NO 0,IPO_FRAME #BASE,POINT2[] " ",TQ_STATE FALSE}
DECL E6POS XP554={X 12675.92788,Y -569.18264,Z 3775.2407,A -83.4604,B -12.81532,C -0.94267,S 2,T 35,E1 -10812.08896,E2 0,E3 0,E4 0,E5 0,E6 0}
; DECL LDAT LCPDATP119={VEL 1,ACC 100,APO_DIST 100,APO_FAC 50.0,ORI_TYP #VAR,CIRC_TYP #BASE,JERK_FAC 50.0}
DECL FDAT FP555={TOOL_NO 0,BASE_NO 0,IPO_FRAME #BASE,POINT2[] " ",TQ_STATE FALSE}
DECL E6POS XP555={X 6034.81499,Y -708.12179,Z 3847.76366,A -102.7078,B 7.77596,C 4.76026,S 2,T 35,E1 -4174.36752,E2 0,E3 0,E4 0,E5 0,E6 0}
; DECL LDAT LCPDATP120={VEL 1,ACC 100,APO_DIST 100,APO_FAC 50.0,ORI_TYP #VAR,CIRC_TYP #BASE,JERK_FAC 50.0}
DECL FDAT FP556={TOOL_NO 0,BASE_NO 0,IPO_FRAME #BASE,POINT2[] " ",TQ_STATE FALSE}
DECL E6POS XP556={X 5808.56571,Y -717.10091,Z 4003.7046,A -102.70779,B 7.77596,C 4.76025,S 2,T 35,E1 -4005.10214,E2 0,E3 0,E4 0,E5 0,E6 0}
; DECL LDAT LCPDATP123={VEL 1,ACC 100,APO_DIST 100,APO_FAC 50.0,ORI_TYP #VAR,CIRC_TYP #BASE,JERK_FAC 50.0}
DECL FDAT FP557={TOOL_NO 0,BASE_NO 0,IPO_FRAME #BASE,POINT2[] " ",TQ_STATE FALSE}
DECL E6POS XP557={X 12607.03936,Y -538.48386,Z 3940.5062,A -83.4604,B -12.81532,C -0.94267,S 2,T 35,E1 -10812.08896,E2 0,E3 0,E4 0,E5 0,E6 0}
; DECL LDAT LCPDATP124={VEL 1,ACC 100,APO_DIST 100,APO_FAC 50.0,ORI_TYP #VAR,CIRC_TYP #BASE,JERK_FAC 50.0}
DECL FDAT FP558={TOOL_NO 0,BASE_NO 0,IPO_FRAME #BASE,POINT2[] " ",TQ_STATE FALSE}
DECL E6POS XP558={X 12329.73693,Y -538.48386,Z 3940.5062,A -83.38777,B -15.32829,C -1.2413,S 2,T 35,E1 -10812.08896,E2 0,E3 0,E4 0,E5 0,E6 0}
; DECL LDAT LCPDATP130={VEL 1,ACC 100,APO_DIST 100,APO_FAC 50.0,ORI_TYP #VAR,CIRC_TYP #BASE,JERK_FAC 50.0}
DECL FDAT FP559={TOOL_NO 0,BASE_NO 0,IPO_FRAME #BASE,POINT2[] " ",TQ_STATE FALSE}
DECL E6POS XP559={X 6035.27715,Y -717.10158,Z 4003.70466,A -106.51042,B 6.34838,C 5.00917,S 2,T 35,E1 -4231.81368,E2 0,E3 0,E4 0,E5 0,E6 0}
; DECL LDAT LCPDATP131={VEL 1,ACC 100,APO_DIST 100,APO_FAC 50.0,ORI_TYP #VAR,CIRC_TYP #BASE,JERK_FAC 50.0}
DECL FDAT FP560={TOOL_NO 0,BASE_NO 0,IPO_FRAME #BASE,POINT2[] " ",TQ_STATE FALSE}
DECL E6POS XP560={X 6001.84737,Y -717.10113,Z 4003.70421,A -106.4599,B 4.5615,C 5.54032,S 2,T 35,E1 -4198.38336,E2 0,E3 0,E4 0,E5 0,E6 0}
; DECL LDAT LCPDATP125={VEL 1,ACC 100,APO_DIST 100,APO_FAC 50.0,ORI_TYP #VAR,CIRC_TYP #BASE,JERK_FAC 50.0}
DECL FDAT FP561={TOOL_NO 0,BASE_NO 0,IPO_FRAME #BASE,POINT2[] " ",TQ_STATE FALSE}
DECL E6POS XP561={X 12327.62864,Y -538.48366,Z 3940.50597,A -87.76623,B -17.49847,C -1.50503,S 2,T 35,E1 -10473.34117,E2 0,E3 0,E4 0,E5 0,E6 0}
; DECL LDAT LCPDATP126={VEL 1,ACC 100,APO_DIST 100,APO_FAC 50.0,ORI_TYP #VAR,CIRC_TYP #BASE,JERK_FAC 50.0}
DECL FDAT FP562={TOOL_NO 0,BASE_NO 0,IPO_FRAME #BASE,POINT2[] " ",TQ_STATE FALSE}
DECL E6POS XP562={X 12344.44126,Y -538.48354,Z 3940.50612,A -92.12133,B -19.55447,C -1.59012,S 2,T 35,E1 -10490.15446,E2 0,E3 0,E4 0,E5 0,E6 0}
; DECL LDAT LCPDATP132={VEL 1,ACC 100,APO_DIST 100,APO_FAC 50.0,ORI_TYP #VAR,CIRC_TYP #BASE,JERK_FAC 50.0}
DECL FDAT FP563={TOOL_NO 0,BASE_NO 0,IPO_FRAME #BASE,POINT2[] " ",TQ_STATE FALSE}
DECL E6POS XP563={X 5984.60315,Y -717.10142,Z 4003.7045,A -107.27293,B 2.66443,C 6.10126,S 2,T 35,E1 -4181.13976,E2 0,E3 0,E4 0,E5 0,E6 0}
; DECL LDAT LCPDATP133={VEL 1,ACC 100,APO_DIST 100,APO_FAC 50.0,ORI_TYP #VAR,CIRC_TYP #BASE,JERK_FAC 50.0}
DECL FDAT FP564={TOOL_NO 0,BASE_NO 0,IPO_FRAME #BASE,POINT2[] " ",TQ_STATE FALSE}
DECL E6POS XP564={X 5959.53065,Y -717.10165,Z 4003.70439,A -107.25516,B 0.74219,C 6.69889,S 2,T 35,E1 -4156.06702,E2 0,E3 0,E4 0,E5 0,E6 0}
; DECL LDAT LCPDATP127={VEL 1,ACC 100,APO_DIST 100,APO_FAC 50.0,ORI_TYP #VAR,CIRC_TYP #BASE,JERK_FAC 50.0}
DECL FDAT FP565={TOOL_NO 0,BASE_NO 0,IPO_FRAME #BASE,POINT2[] " ",TQ_STATE FALSE}
DECL E6POS XP565={X 12327.65948,Y -538.48376,Z 3940.50627,A -96.02004,B -21.56802,C -1.50992,S 2,T 35,E1 -10473.37259,E2 0,E3 0,E4 0,E5 0,E6 0}
; DECL LDAT LCPDATP128={VEL 1,ACC 100,APO_DIST 100,APO_FAC 50.0,ORI_TYP #VAR,CIRC_TYP #BASE,JERK_FAC 50.0}
DECL FDAT FP566={TOOL_NO 0,BASE_NO 0,IPO_FRAME #BASE,POINT2[] " ",TQ_STATE FALSE}
DECL E6POS XP566={X 12434.40962,Y -538.48361,Z 3791.38491,A -100.48203,B -23.59142,C -1.27711,S 2,T 35,E1 -10580.12251,E2 0,E3 0,E4 0,E5 0,E6 0}
; DECL LDAT LCPDATP134={VEL 1,ACC 100,APO_DIST 100,APO_FAC 50.0,ORI_TYP #VAR,CIRC_TYP #BASE,JERK_FAC 50.0}
DECL FDAT FP567={TOOL_NO 0,BASE_NO 0,IPO_FRAME #BASE,POINT2[] " ",TQ_STATE FALSE}
DECL E6POS XP567={X 6027.18413,Y -717.10157,Z 4003.70451,A -108.83879,B -1.2655,C 7.3225,S 2,T 35,E1 -4223.72032,E2 0,E3 0,E4 0,E5 0,E6 0}
; DECL LDAT LCPDATP135={VEL 1,ACC 100,APO_DIST 100,APO_FAC 50.0,ORI_TYP #VAR,CIRC_TYP #BASE,JERK_FAC 50.0}
DECL FDAT FP568={TOOL_NO 0,BASE_NO 0,IPO_FRAME #BASE,POINT2[] " ",TQ_STATE FALSE}
DECL E6POS XP568={X 5994.01853,Y -717.10159,Z 4003.70409,A -109.42003,B -3.44272,C 8.06654,S 2,T 35,E1 -4190.55423,E2 0,E3 0,E4 0,E5 0,E6 0}
; DECL LDAT LCPDATP129={VEL 1,ACC 100,APO_DIST 100,APO_FAC 50.0,ORI_TYP #VAR,CIRC_TYP #BASE,JERK_FAC 50.0}
DECL FDAT FP569={TOOL_NO 0,BASE_NO 0,IPO_FRAME #BASE,POINT2[] " ",TQ_STATE FALSE}
DECL E6POS XP569={X 12525.53957,Y -538.48385,Z 3733.39322,A -103.74147,B -24.12805,C -1.24549,S 2,T 35,E1 -10671.25219,E2 0,E3 0,E4 0,E5 0,E6 0}
; DECL LDAT LCPDATP138={VEL 1,ACC 100,APO_DIST 100,APO_FAC 50.0,ORI_TYP #VAR,CIRC_TYP #BASE,JERK_FAC 50.0}
DECL FDAT FP570={TOOL_NO 0,BASE_NO 0,IPO_FRAME #BASE,POINT2[] " ",TQ_STATE FALSE}
DECL E6POS XP570={X 12409.55634,Y -538.48385,Z 3733.39322,A -103.74147,B -24.12805,C -1.24549,S 2,T 35,E1 -10555.26896,E2 0,E3 0,E4 0,E5 0,E6 0}
; DECL LDAT LCPDATP136={VEL 1,ACC 100,APO_DIST 100,APO_FAC 50.0,ORI_TYP #VAR,CIRC_TYP #BASE,JERK_FAC 50.0}
DECL FDAT FP571={TOOL_NO 0,BASE_NO 0,IPO_FRAME #BASE,POINT2[] " ",TQ_STATE FALSE}
DECL E6POS XP571={X 5960.30101,Y -717.10136,Z 4003.70387,A -109.95564,B -5.51238,C 8.79955,S 2,T 35,E1 -4156.83652,E2 0,E3 0,E4 0,E5 0,E6 0}
; DECL LDAT LCPDATP137={VEL 1,ACC 100,APO_DIST 100,APO_FAC 50.0,ORI_TYP #VAR,CIRC_TYP #BASE,JERK_FAC 50.0}
DECL FDAT FP572={TOOL_NO 0,BASE_NO 0,IPO_FRAME #BASE,POINT2[] " ",TQ_STATE FALSE}
DECL E6POS XP572={X 5959.29294,Y -717.10098,Z 4003.70454,A -110.58224,B -7.77816,C 9.62993,S 2,T 35,E1 -4155.82897,E2 0,E3 0,E4 0,E5 0,E6 0}
; DECL LDAT LCPDATP139={VEL 1,ACC 100,APO_DIST 100,APO_FAC 50.0,ORI_TYP #VAR,CIRC_TYP #BASE,JERK_FAC 50.0}
DECL FDAT FP573={TOOL_NO 0,BASE_NO 0,IPO_FRAME #BASE,POINT2[] " ",TQ_STATE FALSE}
DECL E6POS XP573={X 12666.37592,Y -538.48386,Z 3733.39329,A -110.95703,B -23.34196,C -1.63568,S 2,T 35,E1 -10812.08896,E2 0,E3 0,E4 0,E5 0,E6 0}
; DECL LDAT LCPDATP140={VEL 1,ACC 100,APO_DIST 100,APO_FAC 50.0,ORI_TYP #VAR,CIRC_TYP #BASE,JERK_FAC 50.0}
DECL FDAT FP574={TOOL_NO 0,BASE_NO 0,IPO_FRAME #BASE,POINT2[] " ",TQ_STATE FALSE}
DECL E6POS XP574={X 12666.37592,Y -538.48386,Z 3700.25522,A -113.36831,B -23.34196,C -1.63568,S 2,T 35,E1 -10812.08896,E2 0,E3 0,E4 0,E5 0,E6 0}
; DECL LDAT LCPDATP149={VEL 1,ACC 100,APO_DIST 100,APO_FAC 50.0,ORI_TYP #VAR,CIRC_TYP #BASE,JERK_FAC 50.0}
DECL FDAT FP575={TOOL_NO 0,BASE_NO 0,IPO_FRAME #BASE,POINT2[] " ",TQ_STATE FALSE}
DECL E6POS XP575={X 5916.8006,Y -717.10155,Z 4003.70412,A -110.72224,B -10.13455,C 10.52896,S 2,T 35,E1 -4113.33656,E2 0,E3 0,E4 0,E5 0,E6 0}
; DECL LDAT LCPDATP150={VEL 1,ACC 100,APO_DIST 100,APO_FAC 50.0,ORI_TYP #VAR,CIRC_TYP #BASE,JERK_FAC 50.0}
DECL FDAT FP576={TOOL_NO 0,BASE_NO 0,IPO_FRAME #BASE,POINT2[] " ",TQ_STATE FALSE}
DECL E6POS XP576={X 5875.31565,Y -717.1012,Z 4003.70448,A -110.8879,B -12.32973,C 11.37928,S 2,T 35,E1 -4071.85169,E2 0,E3 0,E4 0,E5 0,E6 0}
; DECL LDAT LCPDATP141={VEL 1,ACC 100,APO_DIST 100,APO_FAC 50.0,ORI_TYP #VAR,CIRC_TYP #BASE,JERK_FAC 50.0}
DECL FDAT FP577={TOOL_NO 0,BASE_NO 0,IPO_FRAME #BASE,POINT2[] " ",TQ_STATE FALSE}
DECL E6POS XP577={X 12666.37592,Y -538.48386,Z 3675.40167,A -115.34787,B -23.34196,C -1.63568,S 2,T 35,E1 -10812.08896,E2 0,E3 0,E4 0,E5 0,E6 0}
; DECL LDAT LCPDATP142={VEL 1,ACC 100,APO_DIST 100,APO_FAC 50.0,ORI_TYP #VAR,CIRC_TYP #BASE,JERK_FAC 50.0}
DECL FDAT FP578={TOOL_NO 0,BASE_NO 0,IPO_FRAME #BASE,POINT2[] " ",TQ_STATE FALSE}
DECL E6POS XP578={X 12666.37592,Y -538.48386,Z 3725.10877,A -117.62399,B -22.31862,C -2.21953,S 2,T 35,E1 -10812.08896,E2 0,E3 0,E4 0,E5 0,E6 0}
; DECL LDAT LCPDATP151={VEL 1,ACC 100,APO_DIST 100,APO_FAC 50.0,ORI_TYP #VAR,CIRC_TYP #BASE,JERK_FAC 50.0}
DECL FDAT FP579={TOOL_NO 0,BASE_NO 0,IPO_FRAME #BASE,POINT2[] " ",TQ_STATE FALSE}
DECL E6POS XP579={X 5898.57722,Y -717.10122,Z 4003.70435,A -112.09203,B -14.38754,C 12.19033,S 2,T 35,E1 -4095.11298,E2 0,E3 0,E4 0,E5 0,E6 0}
; DECL LDAT LCPDATP152={VEL 1,ACC 100,APO_DIST 100,APO_FAC 50.0,ORI_TYP #VAR,CIRC_TYP #BASE,JERK_FAC 50.0}
DECL FDAT FP580={TOOL_NO 0,BASE_NO 0,IPO_FRAME #BASE,POINT2[] " ",TQ_STATE FALSE}
DECL E6POS XP580={X 5854.40488,Y -717.10171,Z 4003.70448,A -112.35649,B -16.71303,C 13.17652,S 2,T 35,E1 -4050.94133,E2 0,E3 0,E4 0,E5 0,E6 0}
; DECL LDAT LCPDATP143={VEL 1,ACC 100,APO_DIST 100,APO_FAC 50.0,ORI_TYP #VAR,CIRC_TYP #BASE,JERK_FAC 50.0}
DECL FDAT FP581={TOOL_NO 0,BASE_NO 0,IPO_FRAME #BASE,POINT2[] " ",TQ_STATE FALSE}
DECL E6POS XP581={X 12666.37592,Y -538.48386,Z 3708.53974,A -119.39266,B -22.0406,C -2.38888,S 2,T 35,E1 -10812.08896,E2 0,E3 0,E4 0,E5 0,E6 0}
; DECL LDAT LCPDATP144={VEL 1,ACC 100,APO_DIST 100,APO_FAC 50.0,ORI_TYP #VAR,CIRC_TYP #BASE,JERK_FAC 50.0}
DECL FDAT FP582={TOOL_NO 0,BASE_NO 0,IPO_FRAME #BASE,POINT2[] " ",TQ_STATE FALSE}
DECL E6POS XP582={X 12666.37592,Y -538.48386,Z 3716.82426,A -121.52366,B -21.70131,C -2.61349,S 2,T 35,E1 -10812.08896,E2 0,E3 0,E4 0,E5 0,E6 0}
; DECL LDAT LCPDATP153={VEL 1,ACC 100,APO_DIST 100,APO_FAC 50.0,ORI_TYP #VAR,CIRC_TYP #BASE,JERK_FAC 50.0}
DECL FDAT FP583={TOOL_NO 0,BASE_NO 0,IPO_FRAME #BASE,POINT2[] " ",TQ_STATE FALSE}
DECL E6POS XP583={X 5865.70091,Y -717.10124,Z 4003.70383,A -113.62634,B -18.80667,C 14.08679,S 2,T 35,E1 -4062.23613,E2 0,E3 0,E4 0,E5 0,E6 0}
; DECL LDAT LCPDATP154={VEL 1,ACC 100,APO_DIST 100,APO_FAC 50.0,ORI_TYP #VAR,CIRC_TYP #BASE,JERK_FAC 50.0}
DECL FDAT FP584={TOOL_NO 0,BASE_NO 0,IPO_FRAME #BASE,POINT2[] " ",TQ_STATE FALSE}
DECL E6POS XP584={X 5786.97193,Y -717.10138,Z 4003.70442,A -113.90846,B -20.59534,C 14.92344,S 2,T 35,E1 -3983.50839,E2 0,E3 0,E4 0,E5 0,E6 0}
; DECL LDAT LCPDATP145={VEL 1,ACC 100,APO_DIST 100,APO_FAC 50.0,ORI_TYP #VAR,CIRC_TYP #BASE,JERK_FAC 50.0}
DECL FDAT FP585={TOOL_NO 0,BASE_NO 0,IPO_FRAME #BASE,POINT2[] " ",TQ_STATE FALSE}
DECL E6POS XP585={X 12666.37592,Y -538.48386,Z 3691.97071,A -122.58569,B -21.70131,C -2.61349,S 2,T 35,E1 -10812.08896,E2 0,E3 0,E4 0,E5 0,E6 0}
; DECL LDAT LCPDATP146={VEL 1,ACC 100,APO_DIST 100,APO_FAC 50.0,ORI_TYP #VAR,CIRC_TYP #BASE,JERK_FAC 50.0}
DECL FDAT FP586={TOOL_NO 0,BASE_NO 0,IPO_FRAME #BASE,POINT2[] " ",TQ_STATE FALSE}
DECL E6POS XP586={X 12666.37592,Y -538.48386,Z 3741.67781,A -124.88801,B -20.60151,C -3.44033,S 2,T 35,E1 -10812.08896,E2 0,E3 0,E4 0,E5 0,E6 0}
; DECL LDAT LCPDATP155={VEL 1,ACC 100,APO_DIST 100,APO_FAC 50.0,ORI_TYP #VAR,CIRC_TYP #BASE,JERK_FAC 50.0}
DECL FDAT FP587={TOOL_NO 0,BASE_NO 0,IPO_FRAME #BASE,POINT2[] " ",TQ_STATE FALSE}
DECL E6POS XP587={X 5766.06143,Y -717.10078,Z 4003.7047,A -114.88478,B -21.82725,C 15.51221,S 2,T 35,E1 -3962.59803,E2 0,E3 0,E4 0,E5 0,E6 0}
; DECL LDAT LCPDATP156={VEL 1,ACC 100,APO_DIST 100,APO_FAC 50.0,ORI_TYP #VAR,CIRC_TYP #BASE,JERK_FAC 50.0}
DECL FDAT FP588={TOOL_NO 0,BASE_NO 0,IPO_FRAME #BASE,POINT2[] " ",TQ_STATE FALSE}
DECL E6POS XP588={X 5671.46198,Y -717.1018,Z 4003.704,A -116.65787,B -23.21109,C 16.21129,S 2,T 35,E1 -3867.99764,E2 0,E3 0,E4 0,E5 0,E6 0}
; DECL LDAT LCPDATP147={VEL 1,ACC 100,APO_DIST 100,APO_FAC 50.0,ORI_TYP #VAR,CIRC_TYP #BASE,JERK_FAC 50.0}
